LIN {X 0,Y 438.323,Z 588.239,A -85,B 0,C 180,E1 -9180.919,E2 -9180.919} C_VEL
LIN {X 0,Y 438.374,Z 587.567,A -85,B 0,C 180,E1 -9181.838,E2 -9181.838} C_VEL
LIN {X 0,Y 438.437,Z 586.498,A -85,B 0,C 180,E1 -9182.756,E2 -9182.756} C_VEL
LIN {X 0,Y 438.522,Z 585.021,A -85,B 0,C 180,E1 -9183.676,E2 -9183.676} C_VEL
LIN {X 0,Y 438.511,Z 581.969,A -85,B 0,C 180,E1 -9185.057,E2 -9185.057} C_VEL
LIN {X 0,Y 438.764,Z 577.857,A -85,B 0,C 180,E1 -9186.438,E2 -9186.438} C_VEL
LIN {X 0,Y 438.979,Z 571.563,A -85,B 0,C 180,E1 -9188.053,E2 -9188.053} C_VEL
LIN {X 0,Y 439.405,Z 564.723,A -85,B 0,C 180,E1 -9189.436,E2 -9189.436} C_VEL
LIN {X 0,Y 439.856,Z 556.275,A -85,B 0,C 180,E1 -9190.821,E2 -9190.821} C_VEL
LIN {X 0,Y 440.371,Z 547.631,A -85,B 0,C 180,E1 -9191.974,E2 -9191.974} C_VEL
LIN {X 0,Y 441.064,Z 537.577,A -85,B 0,C 180,E1 -9193.073,E2 -9193.073} C_VEL
LIN {X 0,Y 441.606,Z 526.721,A -85,B 0,C 180,E1 -9194.046,E2 -9194.046} C_VEL
LIN {X 0,Y 442.181,Z 515.563,A -85,B 0,C 180,E1 -9194.85,E2 -9194.85} C_VEL
LIN {X 0,Y 442.721,Z 503.226,A -85,B 0,C 180,E1 -9195.538,E2 -9195.538} C_VEL
LIN {X 0,Y 441.9,Z 496.755,A -85,B 0,C 180,E1 -9195.864,E2 -9195.864} C_VEL
LIN {X 0,Y 439.098,Z 483.193,A -85,B 0,C 180,E1 -9196.446,E2 -9196.446} C_VEL
LIN {X 0,Y 438.675,Z 481.043,A -85,B 0,C 180,E1 -9196.533,E2 -9196.533} C_VEL
LIN {X 0,Y 438.78,Z 475.256,A -85,B 0,C 180,E1 -9199.655,E2 -9199.655} C_VEL
LIN {X 0,Y 438.918,Z 469.873,A -85,B 0,C 180,E1 -9202.6,E2 -9202.6} C_VEL
LIN {X 0,Y 439.082,Z 464.477,A -85,B 0,C 180,E1 -9205.605,E2 -9205.605} C_VEL
LIN {X 0,Y 439.285,Z 459.037,A -85,B 0,C 180,E1 -9208.683,E2 -9208.683} C_VEL
LIN {X 0,Y 439.494,Z 453.542,A -85,B 0,C 180,E1 -9211.851,E2 -9211.851} C_VEL
LIN {X 0,Y 439.619,Z 449.852,A -85,B 0,C 180,E1 -9214.024,E2 -9214.024} C_VEL
LIN {X 0,Y 439.631,Z 446.118,A -85,B 0,C 180,E1 -9216.263,E2 -9216.263} C_VEL
LIN {X 0,Y 439.451,Z 444.373,A -85,B 0,C 180,E1 -9217.425,E2 -9217.425} C_VEL
LIN {X 0,Y 439.412,Z 444.375,A -85,B 0,C 180,E1 -9219.85,E2 -9219.85} C_VEL
LIN {X 0,Y 439.391,Z 444.378,A -85,B 0,C 180,E1 -9222.627,E2 -9222.627} C_VEL
LIN {X 0,Y 439.408,Z 444.38,A -85,B 0,C 180,E1 -9225.271,E2 -9225.271} C_VEL
LIN {X 0,Y 439.404,Z 444.38,A -85,B 0,C 180,E1 -9228.741,E2 -9228.741} C_VEL
LIN {X 0,Y 439.489,Z 444.514,A -85,B 0,C 180,E1 -9229.915,E2 -9229.915} C_VEL
LIN {X 0,Y 440.084,Z 449.479,A -85,B 0,C 180,E1 -9232.078,E2 -9232.078} C_VEL
LIN {X 0,Y 439.9,Z 456.078,A -85,B 0,C 180,E1 -9234.889,E2 -9234.889} C_VEL
LIN {X 0,Y 439.732,Z 463.121,A -85,B 0,C 180,E1 -9237.895,E2 -9237.895} C_VEL
LIN {X 0,Y 439.576,Z 469.949,A -85,B 0,C 180,E1 -9240.814,E2 -9240.814} C_VEL
LIN {X 0,Y 439.393,Z 476.574,A -85,B 0,C 180,E1 -9243.6,E2 -9243.6} C_VEL
LIN {X 0,Y 439.22,Z 483.432,A -85,B 0,C 180,E1 -9246.419,E2 -9246.419} C_VEL
LIN {X 0,Y 439.101,Z 490.898,A -85,B 0,C 180,E1 -9249.382,E2 -9249.382} C_VEL
LIN {X 0,Y 439.06,Z 492.954,A -85,B 0,C 180,E1 -9250.179,E2 -9250.179} C_VEL
LIN {X 0,Y 442.741,Z 508.655,A -85,B 0,C 180,E1 -9250.733,E2 -9250.733} C_VEL
LIN {X 0,Y 444.731,Z 520.009,A -85,B 0,C 180,E1 -9251.247,E2 -9251.247} C_VEL
LIN {X 0,Y 444.069,Z 533.417,A -85,B 0,C 180,E1 -9251.888,E2 -9251.888} C_VEL
LIN {X 0,Y 443.371,Z 546.477,A -85,B 0,C 180,E1 -9252.709,E2 -9252.709} C_VEL
LIN {X 0,Y 442.529,Z 558.139,A -85,B 0,C 180,E1 -9253.626,E2 -9253.626} C_VEL
LIN {X 0,Y 441.698,Z 569.986,A -85,B 0,C 180,E1 -9254.778,E2 -9254.778} C_VEL
LIN {X 0,Y 441.477,Z 572.611,A -85,B 0,C 180,E1 -9255.067,E2 -9255.067} C_VEL
LIN {X 0,Y 440.46,Z 577.049,A -85,B 0,C 180,E1 -9255.556,E2 -9255.556} C_VEL
LIN {X 0,Y 437.195,Z 584.006,A -85,B 0,C 180,E1 -9256.371,E2 -9256.371} C_VEL
LIN {X 0,Y 433.95,Z 590.468,A -85,B 0,C 180,E1 -9257.26,E2 -9257.26} C_VEL
LIN {X 0,Y 432.977,Z 594.128,A -85,B 0,C 180,E1 -9257.858,E2 -9257.858} C_VEL
LIN {X 0,Y 432.269,Z 602.417,A -85,B 0,C 180,E1 -9259.46,E2 -9259.46} C_VEL
LIN {X 0,Y 431.823,Z 609.29,A -85,B 0,C 180,E1 -9261.104,E2 -9261.104} C_VEL
LIN {X 0,Y 431.475,Z 615.452,A -85,B 0,C 180,E1 -9262.982,E2 -9262.982} C_VEL
LIN {X 0,Y 431.38,Z 618.954,A -85,B 0,C 180,E1 -9264.389,E2 -9264.389} C_VEL
LIN {X 0,Y 431.187,Z 622.376,A -85,B 0,C 180,E1 -9266.261,E2 -9266.261} C_VEL
LIN {X 0,Y 431.198,Z 624.413,A -85,B 0,C 180,E1 -9268.131,E2 -9268.131} C_VEL
LIN {X 0,Y 431.143,Z 625.119,A -85,B 0,C 180,E1 -9269.999,E2 -9269.999} C_VEL
LIN {X 0,Y 431.197,Z 624.493,A -85,B 0,C 180,E1 -9271.867,E2 -9271.867} C_VEL
LIN {X 0,Y 431.186,Z 622.523,A -85,B 0,C 180,E1 -9273.737,E2 -9273.737} C_VEL
LIN {X 0,Y 431.379,Z 619.168,A -85,B 0,C 180,E1 -9275.608,E2 -9275.608} C_VEL
LIN {X 0,Y 431.53,Z 614.329,A -85,B 0,C 180,E1 -9277.485,E2 -9277.485} C_VEL
LIN {X 0,Y 431.922,Z 607.864,A -85,B 0,C 180,E1 -9279.363,E2 -9279.363} C_VEL
LIN {X 0,Y 432.355,Z 600.66,A -85,B 0,C 180,E1 -9281.01,E2 -9281.01} C_VEL
LIN {X 0,Y 433.045,Z 593.096,A -85,B 0,C 180,E1 -9282.416,E2 -9282.416} C_VEL
LIN {X 0,Y 433.619,Z 584.184,A -85,B 0,C 180,E1 -9283.806,E2 -9283.806} C_VEL
LIN {X 0,Y 434.507,Z 573.995,A -85,B 0,C 180,E1 -9285.117,E2 -9285.117} C_VEL
LIN {X 0,Y 435.336,Z 562.966,A -85,B 0,C 180,E1 -9286.289,E2 -9286.289} C_VEL
LIN {X 0,Y 436.298,Z 550.821,A -85,B 0,C 180,E1 -9287.336,E2 -9287.336} C_VEL
LIN {X 0,Y 437.081,Z 538.305,A -85,B 0,C 180,E1 -9288.206,E2 -9288.206} C_VEL
LIN {X 0,Y 437.756,Z 524.511,A -85,B 0,C 180,E1 -9288.949,E2 -9288.949} C_VEL
LIN {X 0,Y 437.768,Z 519.177,A -85,B 0,C 180,E1 -9289.191,E2 -9289.191} C_VEL
LIN {X 0,Y 434.917,Z 504.739,A -85,B 0,C 180,E1 -9289.836,E2 -9289.836} C_VEL
LIN {X 0,Y 432.014,Z 492.976,A -85,B 0,C 180,E1 -9290.246,E2 -9290.246} C_VEL
LIN {X 0,Y 432.131,Z 486.1,A -85,B 0,C 180,E1 -9292.973,E2 -9292.973} C_VEL
LIN {X 0,Y 432.305,Z 478.646,A -85,B 0,C 180,E1 -9296.035,E2 -9296.035} C_VEL
LIN {X 0,Y 432.512,Z 472.428,A -85,B 0,C 180,E1 -9298.662,E2 -9298.662} C_VEL
LIN {X 0,Y 432.691,Z 465.079,A -85,B 0,C 180,E1 -9301.841,E2 -9301.841} C_VEL
LIN {X 0,Y 432.919,Z 457.333,A -85,B 0,C 180,E1 -9305.183,E2 -9305.183} C_VEL
LIN {X 0,Y 433.104,Z 450.634,A -85,B 0,C 180,E1 -9308.068,E2 -9308.068} C_VEL
LIN {X 0,Y 432.706,Z 446.81,A -85,B 0,C 180,E1 -9309.743,E2 -9309.743} C_VEL
LIN {X 0,Y 432.411,Z 445.251,A -85,B 0,C 180,E1 -9310.442,E2 -9310.442} C_VEL
LIN {X 0,Y 432.359,Z 445.256,A -85,B 0,C 180,E1 -9313.054,E2 -9313.054} C_VEL
LIN {X 0,Y 432.371,Z 445.254,A -85,B 0,C 180,E1 -9315.657,E2 -9315.657} C_VEL
LIN {X 0,Y 432.366,Z 445.254,A -85,B 0,C 180,E1 -9318.391,E2 -9318.391} C_VEL
LIN {X 0,Y 432.344,Z 445.254,A -85,B 0,C 180,E1 -9321.851,E2 -9321.851} C_VEL
LIN {X 0,Y 432.332,Z 445.253,A -85,B 0,C 180,E1 -9325.322,E2 -9325.322} C_VEL
LIN {X 0,Y 432.321,Z 445.253,A -85,B 0,C 180,E1 -9328.654,E2 -9328.654} C_VEL
LIN {X 0,Y 432.375,Z 445.251,A -85,B 0,C 180,E1 -9331.876,E2 -9331.876} C_VEL
LIN {X 0,Y 432.342,Z 445.256,A -85,B 0,C 180,E1 -9334.998,E2 -9334.998} C_VEL
LIN {X 0,Y 432.367,Z 445.244,A -85,B 0,C 180,E1 -9338.046,E2 -9338.046} C_VEL
LIN {X 0,Y 432.376,Z 445.25,A -85,B 0,C 180,E1 -9341.029,E2 -9341.029} C_VEL
LIN {X 0,Y 432.432,Z 445.246,A -85,B 0,C 180,E1 -9343.961,E2 -9343.961} C_VEL
LIN {X 0,Y 432.471,Z 445.236,A -85,B 0,C 180,E1 -9347.804,E2 -9347.804} C_VEL
LIN {X 0,Y 432.481,Z 445.234,A -85,B 0,C 180,E1 -9351.59,E2 -9351.59} C_VEL
LIN {X 0,Y 432.594,Z 445.223,A -85,B 0,C 180,E1 -9354.406,E2 -9354.406} C_VEL
LIN {X 0,Y 432.596,Z 445.221,A -85,B 0,C 180,E1 -9358.138,E2 -9358.138} C_VEL
LIN {X 0,Y 432.724,Z 445.207,A -85,B 0,C 180,E1 -9360,E2 -9360} C_VEL
LIN {X 0,Y 432.596,Z 445.214,A -85,B 0,C 180,E1 -9362.794,E2 -9362.794} C_VEL
LIN {X 0,Y 432.562,Z 445.231,A -85,B 0,C 180,E1 -9366.53,E2 -9366.53} C_VEL
LIN {X 0,Y 432.435,Z 445.24,A -85,B 0,C 180,E1 -9369.353,E2 -9369.353} C_VEL
LIN {X 0,Y 432.434,Z 445.24,A -85,B 0,C 180,E1 -9372.812,E2 -9372.812} C_VEL
LIN {X 0,Y 432.401,Z 445.242,A -85,B 0,C 180,E1 -9376.479,E2 -9376.479} C_VEL
LIN {X 0,Y 432.329,Z 445.256,A -85,B 0,C 180,E1 -9379.961,E2 -9379.961} C_VEL
LIN {X 0,Y 432.309,Z 445.257,A -85,B 0,C 180,E1 -9382.965,E2 -9382.965} C_VEL
LIN {X 0,Y 432.354,Z 445.253,A -85,B 0,C 180,E1 -9386.033,E2 -9386.033} C_VEL
LIN {X 0,Y 432.343,Z 445.257,A -85,B 0,C 180,E1 -9389.187,E2 -9389.187} C_VEL
LIN {X 0,Y 432.316,Z 445.262,A -85,B 0,C 180,E1 -9392.294,E2 -9392.294} C_VEL
LIN {X 0,Y 432.332,Z 445.257,A -85,B 0,C 180,E1 -9394.678,E2 -9394.678} C_VEL
LIN {X 0,Y 432.345,Z 445.254,A -85,B 0,C 180,E1 -9398.149,E2 -9398.149} C_VEL
LIN {X 0,Y 432.365,Z 445.251,A -85,B 0,C 180,E1 -9401.609,E2 -9401.609} C_VEL
LIN {X 0,Y 432.371,Z 445.255,A -85,B 0,C 180,E1 -9404.343,E2 -9404.343} C_VEL
LIN {X 0,Y 432.36,Z 445.255,A -85,B 0,C 180,E1 -9408.394,E2 -9408.394} C_VEL
LIN {X 0,Y 432.406,Z 445.352,A -85,B 0,C 180,E1 -9410.921,E2 -9410.921} C_VEL
LIN {X 0,Y 433.952,Z 453.805,A -85,B 0,C 180,E1 -9414.338,E2 -9414.338} C_VEL
LIN {X 0,Y 435.07,Z 459.857,A -85,B 0,C 180,E1 -9416.688,E2 -9416.688} C_VEL
LIN {X 0,Y 434.697,Z 466.214,A -85,B 0,C 180,E1 -9418.968,E2 -9418.968} C_VEL
LIN {X 0,Y 433.899,Z 476.402,A -85,B 0,C 180,E1 -9422.51,E2 -9422.51} C_VEL
LIN {X 0,Y 433.157,Z 486.96,A -85,B 0,C 180,E1 -9426.071,E2 -9426.071} C_VEL
LIN {X 0,Y 432.552,Z 497.544,A -85,B 0,C 180,E1 -9429.555,E2 -9429.555} C_VEL
LIN {X 0,Y 432.493,Z 499.108,A -85,B 0,C 180,E1 -9430.064,E2 -9430.064} C_VEL
LIN {X 0,Y 435.543,Z 514.142,A -85,B 0,C 180,E1 -9430.548,E2 -9430.548} C_VEL
LIN {X 0,Y 437.339,Z 527.333,A -85,B 0,C 180,E1 -9431.106,E2 -9431.106} C_VEL
LIN {X 0,Y 436.738,Z 540.749,A -85,B 0,C 180,E1 -9431.751,E2 -9431.751} C_VEL
LIN {X 0,Y 436.051,Z 553.155,A -85,B 0,C 180,E1 -9432.533,E2 -9432.533} C_VEL
LIN {X 0,Y 435.2,Z 565,A -85,B 0,C 180,E1 -9433.465,E2 -9433.465} C_VEL
LIN {X 0,Y 434.267,Z 576.984,A -85,B 0,C 180,E1 -9434.634,E2 -9434.634} C_VEL
LIN {X 0,Y 433.482,Z 587.773,A -85,B 0,C 180,E1 -9435.926,E2 -9435.926} C_VEL
LIN {X 0,Y 432.889,Z 595.988,A -85,B 0,C 180,E1 -9437.103,E2 -9437.103} C_VEL
LIN {X 0,Y 432.407,Z 604.261,A -85,B 0,C 180,E1 -9438.517,E2 -9438.517} C_VEL
LIN {X 0,Y 431.889,Z 612.153,A -85,B 0,C 180,E1 -9440.163,E2 -9440.163} C_VEL
LIN {X 0,Y 431.566,Z 617.671,A -85,B 0,C 180,E1 -9441.573,E2 -9441.573} C_VEL
LIN {X 0,Y 431.374,Z 623.442,A -85,B 0,C 180,E1 -9443.453,E2 -9443.453} C_VEL
LIN {X 0,Y 431.256,Z 627.631,A -85,B 0,C 180,E1 -9445.327,E2 -9445.327} C_VEL
LIN {X 0,Y 431.239,Z 630.364,A -85,B 0,C 180,E1 -9447.199,E2 -9447.199} C_VEL
LIN {X 0,Y 431.193,Z 631.718,A -85,B 0,C 180,E1 -9449.067,E2 -9449.067} C_VEL
LIN {X 0,Y 431.194,Z 631.716,A -85,B 0,C 180,E1 -9450.935,E2 -9450.935} C_VEL
LIN {X 0,Y 431.24,Z 630.356,A -85,B 0,C 180,E1 -9452.804,E2 -9452.804} C_VEL
LIN {X 0,Y 431.259,Z 627.62,A -85,B 0,C 180,E1 -9454.675,E2 -9454.675} C_VEL
LIN {X 0,Y 431.375,Z 623.432,A -85,B 0,C 180,E1 -9456.55,E2 -9456.55} C_VEL
LIN {X 0,Y 431.573,Z 617.658,A -85,B 0,C 180,E1 -9458.429,E2 -9458.429} C_VEL
LIN {X 0,Y 431.911,Z 611.127,A -85,B 0,C 180,E1 -9460.075,E2 -9460.075} C_VEL
LIN {X 0,Y 432.468,Z 602.992,A -85,B 0,C 180,E1 -9461.722,E2 -9461.722} C_VEL
LIN {X 0,Y 432.969,Z 594.448,A -85,B 0,C 180,E1 -9463.136,E2 -9463.136} C_VEL
LIN {X 0,Y 433.797,Z 584.064,A -85,B 0,C 180,E1 -9464.545,E2 -9464.545} C_VEL
LIN {X 0,Y 434.595,Z 573.594,A -85,B 0,C 180,E1 -9465.717,E2 -9465.717} C_VEL
LIN {X 0,Y 435.399,Z 562.163,A -85,B 0,C 180,E1 -9466.771,E2 -9466.771} C_VEL
LIN {X 0,Y 436.238,Z 549.602,A -85,B 0,C 180,E1 -9467.704,E2 -9467.704} C_VEL
LIN {X 0,Y 436.985,Z 535.644,A -85,B 0,C 180,E1 -9468.513,E2 -9468.513} C_VEL
LIN {X 0,Y 437.262,Z 525.796,A -85,B 0,C 180,E1 -9468.957,E2 -9468.957} C_VEL
LIN {X 0,Y 434.367,Z 506.853,A -85,B 0,C 180,E1 -9469.766,E2 -9469.766} C_VEL
LIN {X 0,Y 432.545,Z 498.491,A -85,B 0,C 180,E1 -9470.119,E2 -9470.119} C_VEL
LIN {X 0,Y 433.089,Z 488.854,A -85,B 0,C 180,E1 -9473.428,E2 -9473.428} C_VEL
LIN {X 0,Y 433.826,Z 480.569,A -85,B 0,C 180,E1 -9476.456,E2 -9476.456} C_VEL
LIN {X 0,Y 434.747,Z 472.778,A -85,B 0,C 180,E1 -9479.554,E2 -9479.554} C_VEL
LIN {X 0,Y 435.75,Z 466.846,A -85,B 0,C 180,E1 -9482.158,E2 -9482.158} C_VEL
LIN {X 0,Y 435.961,Z 463.596,A -85,B 0,C 180,E1 -9483.792,E2 -9483.792} C_VEL
LIN {X 0,Y 435.29,Z 459.741,A -85,B 0,C 180,E1 -9486.169,E2 -9486.169} C_VEL
LIN {X 0,Y 434.63,Z 456.055,A -85,B 0,C 180,E1 -9489.098,E2 -9489.098} C_VEL
LIN {X 0,Y 434.129,Z 453.741,A -85,B 0,C 180,E1 -9491.868,E2 -9491.868} C_VEL
LIN {X 0,Y 433.839,Z 452.608,A -85,B 0,C 180,E1 -9494.538,E2 -9494.538} C_VEL
LIN {X 0,Y 433.817,Z 452.479,A -85,B 0,C 180,E1 -9497.124,E2 -9497.124} C_VEL
LIN {X 0,Y 433.888,Z 453.237,A -85,B 0,C 180,E1 -9499.616,E2 -9499.616} C_VEL
LIN {X 0,Y 434.126,Z 454.981,A -85,B 0,C 180,E1 -9502.492,E2 -9502.492} C_VEL
LIN {X 0,Y 434.122,Z 456.599,A -85,B 0,C 180,E1 -9504.352,E2 -9504.352} C_VEL
LIN {X 0,Y 433.574,Z 460.031,A -85,B 0,C 180,E1 -9507.448,E2 -9507.448} C_VEL
LIN {X 0,Y 433.215,Z 463.025,A -85,B 0,C 180,E1 -9509.807,E2 -9509.807} C_VEL
LIN {X 0,Y 432.764,Z 467.893,A -85,B 0,C 180,E1 -9513.278,E2 -9513.278} C_VEL
LIN {X 0,Y 432.348,Z 473.626,A -85,B 0,C 180,E1 -9517.037,E2 -9517.037} C_VEL
LIN {X 0,Y 432.09,Z 478.453,A -85,B 0,C 180,E1 -9520.028,E2 -9520.028} C_VEL
LIN {X 0,Y 431.907,Z 482.91,A -85,B 0,C 180,E1 -9522.694,E2 -9522.694} C_VEL
LIN {X 0,Y 435.601,Z 496.817,A -85,B 0,C 180,E1 -9523.46,E2 -9523.46} C_VEL
LIN {X 0,Y 436.8,Z 504.591,A -85,B 0,C 180,E1 -9523.923,E2 -9523.923} C_VEL
LIN {X 0,Y 436.083,Z 517.539,A -85,B 0,C 180,E1 -9524.698,E2 -9524.698} C_VEL
LIN {X 0,Y 435.299,Z 529.583,A -85,B 0,C 180,E1 -9525.632,E2 -9525.632} C_VEL
LIN {X 0,Y 434.468,Z 541.516,A -85,B 0,C 180,E1 -9526.792,E2 -9526.792} C_VEL
LIN {X 0,Y 433.621,Z 552.042,A -85,B 0,C 180,E1 -9528.074,E2 -9528.074} C_VEL
LIN {X 0,Y 432.957,Z 561.383,A -85,B 0,C 180,E1 -9529.478,E2 -9529.478} C_VEL
LIN {X 0,Y 432.448,Z 568.909,A -85,B 0,C 180,E1 -9530.883,E2 -9530.883} C_VEL
LIN {X 0,Y 431.935,Z 575.885,A -85,B 0,C 180,E1 -9532.521,E2 -9532.521} C_VEL
LIN {X 0,Y 431.726,Z 580.518,A -85,B 0,C 180,E1 -9533.926,E2 -9533.926} C_VEL
LIN {X 0,Y 431.505,Z 584.058,A -85,B 0,C 180,E1 -9535.329,E2 -9535.329} C_VEL
LIN {X 0,Y 431.496,Z 585.867,A -85,B 0,C 180,E1 -9536.265,E2 -9536.265} C_VEL
LIN {X 0,Y 431.379,Z 587.216,A -85,B 0,C 180,E1 -9537.199,E2 -9537.199} C_VEL
LIN {X 0,Y 431.264,Z 588.713,A -85,B 0,C 180,E1 -9539.066,E2 -9539.066} C_VEL
LIN {X 0,Y 431.248,Z 588.865,A -85,B 0,C 180,E1 -9540,E2 -9540} C_VEL
LIN {X 0,Y 431.236,Z 588.576,A -85,B 0,C 180,E1 -9540.934,E2 -9540.934} C_VEL
LIN {X 0,Y 431.294,Z 587.886,A -85,B 0,C 180,E1 -9541.868,E2 -9541.868} C_VEL
LIN {X 0,Y 431.369,Z 586.801,A -85,B 0,C 180,E1 -9542.802,E2 -9542.802} C_VEL
LIN {X 0,Y 431.444,Z 585.302,A -85,B 0,C 180,E1 -9543.736,E2 -9543.736} C_VEL
LIN {X 0,Y 431.453,Z 582.218,A -85,B 0,C 180,E1 -9545.14,E2 -9545.14} C_VEL
LIN {X 0,Y 431.667,Z 577.501,A -85,B 0,C 180,E1 -9546.708,E2 -9546.708} C_VEL
LIN {X 0,Y 431.997,Z 570.685,A -85,B 0,C 180,E1 -9548.419,E2 -9548.419} C_VEL
LIN {X 0,Y 432.418,Z 563.565,A -85,B 0,C 180,E1 -9549.826,E2 -9549.826} C_VEL
LIN {X 0,Y 432.947,Z 554.694,A -85,B 0,C 180,E1 -9551.233,E2 -9551.233} C_VEL
LIN {X 0,Y 433.646,Z 544.694,A -85,B 0,C 180,E1 -9552.519,E2 -9552.519} C_VEL
LIN {X 0,Y 434.322,Z 534.739,A -85,B 0,C 180,E1 -9553.56,E2 -9553.56} C_VEL
LIN {X 0,Y 434.857,Z 523.63,A -85,B 0,C 180,E1 -9554.508,E2 -9554.508} C_VEL
LIN {X 0,Y 435.495,Z 511.594,A -85,B 0,C 180,E1 -9555.323,E2 -9555.323} C_VEL
LIN {X 0,Y 435.692,Z 501.751,A -85,B 0,C 180,E1 -9555.856,E2 -9555.856} C_VEL
LIN {X 0,Y 433.167,Z 488.577,A -85,B 0,C 180,E1 -9556.498,E2 -9556.498} C_VEL
LIN {X 0,Y 431.592,Z 481.162,A -85,B 0,C 180,E1 -9556.811,E2 -9556.811} C_VEL
LIN {X 0,Y 431.713,Z 475.33,A -85,B 0,C 180,E1 -9559.991,E2 -9559.991} C_VEL
LIN {X 0,Y 431.886,Z 469.92,A -85,B 0,C 180,E1 -9562.989,E2 -9562.989} C_VEL
LIN {X 0,Y 432.119,Z 463.61,A -85,B 0,C 180,E1 -9566.551,E2 -9566.551} C_VEL
LIN {X 0,Y 432.378,Z 457.191,A -85,B 0,C 180,E1 -9570.257,E2 -9570.257} C_VEL
LIN {X 0,Y 432.551,Z 451.642,A -85,B 0,C 180,E1 -9573.534,E2 -9573.534} C_VEL
LIN {X 0,Y 432.62,Z 447.905,A -85,B 0,C 180,E1 -9575.791,E2 -9575.791} C_VEL
LIN {X 0,Y 432.415,Z 445.248,A -85,B 0,C 180,E1 -9577.517,E2 -9577.517} C_VEL
LIN {X 0,Y 432.332,Z 445.257,A -85,B 0,C 180,E1 -9580.56,E2 -9580.56} C_VEL
LIN {X 0,Y 432.329,Z 445.259,A -85,B 0,C 180,E1 -9583.06,E2 -9583.06} C_VEL
LIN {X 0,Y 432.339,Z 445.26,A -85,B 0,C 180,E1 -9585.664,E2 -9585.664} C_VEL
LIN {X 0,Y 432.372,Z 445.257,A -85,B 0,C 180,E1 -9588.392,E2 -9588.392} C_VEL
LIN {X 0,Y 432.437,Z 445.4,A -85,B 0,C 180,E1 -9589.736,E2 -9589.736} C_VEL
LIN {X 0,Y 433.058,Z 450.329,A -85,B 0,C 180,E1 -9591.924,E2 -9591.924} C_VEL
LIN {X 0,Y 432.897,Z 457.046,A -85,B 0,C 180,E1 -9594.813,E2 -9594.813} C_VEL
LIN {X 0,Y 432.733,Z 463.568,A -85,B 0,C 180,E1 -9597.622,E2 -9597.622} C_VEL
LIN {X 0,Y 432.541,Z 470.988,A -85,B 0,C 180,E1 -9600.826,E2 -9600.826} C_VEL
LIN {X 0,Y 432.375,Z 477.007,A -85,B 0,C 180,E1 -9603.38,E2 -9603.38} C_VEL
LIN {X 0,Y 432.169,Z 484.596,A -85,B 0,C 180,E1 -9606.519,E2 -9606.519} C_VEL
LIN {X 0,Y 432.033,Z 492.151,A -85,B 0,C 180,E1 -9609.528,E2 -9609.528} C_VEL
LIN {X 0,Y 432.031,Z 492.973,A -85,B 0,C 180,E1 -9609.849,E2 -9609.849} C_VEL
LIN {X 0,Y 435.634,Z 508.113,A -85,B 0,C 180,E1 -9610.39,E2 -9610.39} C_VEL
LIN {X 0,Y 437.971,Z 520.738,A -85,B 0,C 180,E1 -9610.976,E2 -9610.976} C_VEL
LIN {X 0,Y 437.275,Z 534.382,A -85,B 0,C 180,E1 -9611.649,E2 -9611.649} C_VEL
LIN {X 0,Y 436.59,Z 546.521,A -85,B 0,C 180,E1 -9612.432,E2 -9612.432} C_VEL
LIN {X 0,Y 435.703,Z 558.186,A -85,B 0,C 180,E1 -9613.362,E2 -9613.362} C_VEL
LIN {X 0,Y 434.831,Z 570.037,A -85,B 0,C 180,E1 -9614.532,E2 -9614.532} C_VEL
LIN {X 0,Y 433.999,Z 579.862,A -85,B 0,C 180,E1 -9615.702,E2 -9615.702} C_VEL
LIN {X 0,Y 433.258,Z 589.648,A -85,B 0,C 180,E1 -9617.111,E2 -9617.111} C_VEL
LIN {X 0,Y 432.977,Z 594.128,A -85,B 0,C 180,E1 -9617.858,E2 -9617.858} C_VEL
LIN {X 0,Y 431.992,Z 597.662,A -85,B 0,C 180,E1 -9618.478,E2 -9618.478} C_VEL
LIN {X 0,Y 428.725,Z 603.037,A -85,B 0,C 180,E1 -9619.5,E2 -9619.5} C_VEL
LIN {X 0,Y 425.547,Z 607.883,A -85,B 0,C 180,E1 -9620.58,E2 -9620.58} C_VEL
LIN {X 0,Y 424.709,Z 610.507,A -85,B 0,C 180,E1 -9621.281,E2 -9621.281} C_VEL
LIN {X 0,Y 424.413,Z 615.508,A -85,B 0,C 180,E1 -9622.865,E2 -9622.865} C_VEL
LIN {X 0,Y 424.288,Z 619.01,A -85,B 0,C 180,E1 -9624.295,E2 -9624.295} C_VEL
LIN {X 0,Y 424.098,Z 622.432,A -85,B 0,C 180,E1 -9626.198,E2 -9626.198} C_VEL
LIN {X 0,Y 424.124,Z 624.469,A -85,B 0,C 180,E1 -9628.1,E2 -9628.1} C_VEL
LIN {X 0,Y 424.061,Z 625.174,A -85,B 0,C 180,E1 -9629.999,E2 -9629.999} C_VEL
LIN {X 0,Y 424.123,Z 624.548,A -85,B 0,C 180,E1 -9631.898,E2 -9631.898} C_VEL
LIN {X 0,Y 424.097,Z 622.578,A -85,B 0,C 180,E1 -9633.799,E2 -9633.799} C_VEL
LIN {X 0,Y 424.284,Z 619.222,A -85,B 0,C 180,E1 -9635.703,E2 -9635.703} C_VEL
LIN {X 0,Y 424.466,Z 614.382,A -85,B 0,C 180,E1 -9637.61,E2 -9637.61} C_VEL
LIN {X 0,Y 424.891,Z 607.916,A -85,B 0,C 180,E1 -9639.52,E2 -9639.52} C_VEL
LIN {X 0,Y 425.361,Z 600.71,A -85,B 0,C 180,E1 -9641.193,E2 -9641.193} C_VEL
LIN {X 0,Y 426.075,Z 593.19,A -85,B 0,C 180,E1 -9642.615,E2 -9642.615} C_VEL
LIN {X 0,Y 426.689,Z 584.072,A -85,B 0,C 180,E1 -9644.059,E2 -9644.059} C_VEL
LIN {X 0,Y 427.625,Z 574.038,A -85,B 0,C 180,E1 -9645.366,E2 -9645.366} C_VEL
LIN {X 0,Y 428.527,Z 563.005,A -85,B 0,C 180,E1 -9646.555,E2 -9646.555} C_VEL
LIN {X 0,Y 429.521,Z 550.855,A -85,B 0,C 180,E1 -9647.619,E2 -9647.619} C_VEL
LIN {X 0,Y 430.299,Z 539,A -85,B 0,C 180,E1 -9648.46,E2 -9648.46} C_VEL
LIN {X 0,Y 430.933,Z 526.371,A -85,B 0,C 180,E1 -9649.169,E2 -9649.169} C_VEL
LIN {X 0,Y 431.06,Z 520.429,A -85,B 0,C 180,E1 -9649.448,E2 -9649.448} C_VEL
LIN {X 0,Y 428.263,Z 506.294,A -85,B 0,C 180,E1 -9650.11,E2 -9650.11} C_VEL
LIN {X 0,Y 424.986,Z 492.957,A -85,B 0,C 180,E1 -9650.604,E2 -9650.604} C_VEL
LIN {X 0,Y 425.145,Z 484.759,A -85,B 0,C 180,E1 -9653.89,E2 -9653.89} C_VEL
LIN {X 0,Y 425.365,Z 477.677,A -85,B 0,C 180,E1 -9656.848,E2 -9656.848} C_VEL
LIN {X 0,Y 425.607,Z 469.802,A -85,B 0,C 180,E1 -9660.24,E2 -9660.24} C_VEL
LIN {X 0,Y 425.868,Z 460.928,A -85,B 0,C 180,E1 -9664.13,E2 -9664.13} C_VEL
LIN {X 0,Y 426.114,Z 452.807,A -85,B 0,C 180,E1 -9667.657,E2 -9667.657} C_VEL
LIN {X 0,Y 425.823,Z 448.492,A -85,B 0,C 180,E1 -9669.567,E2 -9669.567} C_VEL
LIN {X 0,Y 425.336,Z 446.133,A -85,B 0,C 180,E1 -9670.682,E2 -9670.682} C_VEL
LIN {X 0,Y 425.312,Z 446.132,A -85,B 0,C 180,E1 -9673.947,E2 -9673.947} C_VEL
LIN {X 0,Y 425.325,Z 446.133,A -85,B 0,C 180,E1 -9677.353,E2 -9677.353} C_VEL
LIN {X 0,Y 425.316,Z 446.132,A -85,B 0,C 180,E1 -9681.103,E2 -9681.103} C_VEL
LIN {X 0,Y 425.292,Z 446.135,A -85,B 0,C 180,E1 -9684.663,E2 -9684.663} C_VEL
LIN {X 0,Y 425.264,Z 446.139,A -85,B 0,C 180,E1 -9688.073,E2 -9688.073} C_VEL
LIN {X 0,Y 425.328,Z 446.131,A -85,B 0,C 180,E1 -9691.368,E2 -9691.368} C_VEL
LIN {X 0,Y 425.286,Z 446.131,A -85,B 0,C 180,E1 -9694.554,E2 -9694.554} C_VEL
LIN {X 0,Y 425.31,Z 446.122,A -85,B 0,C 180,E1 -9697.719,E2 -9697.719} C_VEL
LIN {X 0,Y 425.355,Z 446.127,A -85,B 0,C 180,E1 -9700.704,E2 -9700.704} C_VEL
LIN {X 0,Y 425.388,Z 446.124,A -85,B 0,C 180,E1 -9703.688,E2 -9703.688} C_VEL
LIN {X 0,Y 425.42,Z 446.116,A -85,B 0,C 180,E1 -9707.598,E2 -9707.598} C_VEL
LIN {X 0,Y 425.432,Z 446.112,A -85,B 0,C 180,E1 -9711.45,E2 -9711.45} C_VEL
LIN {X 0,Y 425.569,Z 446.099,A -85,B 0,C 180,E1 -9714.313,E2 -9714.313} C_VEL
LIN {X 0,Y 425.565,Z 446.097,A -85,B 0,C 180,E1 -9718.107,E2 -9718.107} C_VEL
LIN {X 0,Y 425.694,Z 446.083,A -85,B 0,C 180,E1 -9720,E2 -9720} C_VEL
LIN {X 0,Y 425.548,Z 446.09,A -85,B 0,C 180,E1 -9722.84,E2 -9722.84} C_VEL
LIN {X 0,Y 425.52,Z 446.107,A -85,B 0,C 180,E1 -9726.639,E2 -9726.639} C_VEL
LIN {X 0,Y 425.394,Z 446.115,A -85,B 0,C 180,E1 -9729.509,E2 -9729.509} C_VEL
LIN {X 0,Y 425.393,Z 446.117,A -85,B 0,C 180,E1 -9732.911,E2 -9732.911} C_VEL
LIN {X 0,Y 425.35,Z 446.118,A -85,B 0,C 180,E1 -9736.605,E2 -9736.605} C_VEL
LIN {X 0,Y 425.318,Z 446.127,A -85,B 0,C 180,E1 -9739.636,E2 -9739.636} C_VEL
LIN {X 0,Y 425.297,Z 446.133,A -85,B 0,C 180,E1 -9743.366,E2 -9743.366} C_VEL
LIN {X 0,Y 425.339,Z 446.129,A -85,B 0,C 180,E1 -9746.845,E2 -9746.845} C_VEL
LIN {X 0,Y 425.309,Z 446.131,A -85,B 0,C 180,E1 -9749.718,E2 -9749.718} C_VEL
LIN {X 0,Y 425.273,Z 446.135,A -85,B 0,C 180,E1 -9753.049,E2 -9753.049} C_VEL
LIN {X 0,Y 425.276,Z 446.137,A -85,B 0,C 180,E1 -9755.93,E2 -9755.93} C_VEL
LIN {X 0,Y 425.305,Z 446.133,A -85,B 0,C 180,E1 -9759.047,E2 -9759.047} C_VEL
LIN {X 0,Y 425.324,Z 446.133,A -85,B 0,C 180,E1 -9762.647,E2 -9762.647} C_VEL
LIN {X 0,Y 425.287,Z 446.134,A -85,B 0,C 180,E1 -9765.283,E2 -9765.283} C_VEL
LIN {X 0,Y 425.298,Z 446.135,A -85,B 0,C 180,E1 -9768.626,E2 -9768.626} C_VEL
LIN {X 0,Y 425.348,Z 446.207,A -85,B 0,C 180,E1 -9770.594,E2 -9770.594} C_VEL
LIN {X 0,Y 426.783,Z 453.952,A -85,B 0,C 180,E1 -9773.794,E2 -9773.794} C_VEL
LIN {X 0,Y 428.053,Z 460.799,A -85,B 0,C 180,E1 -9776.509,E2 -9776.509} C_VEL
LIN {X 0,Y 427.859,Z 465.644,A -85,B 0,C 180,E1 -9778.291,E2 -9778.291} C_VEL
LIN {X 0,Y 427.081,Z 474.652,A -85,B 0,C 180,E1 -9781.498,E2 -9781.498} C_VEL
LIN {X 0,Y 426.379,Z 483.677,A -85,B 0,C 180,E1 -9784.626,E2 -9784.626} C_VEL
LIN {X 0,Y 425.787,Z 492.718,A -85,B 0,C 180,E1 -9787.69,E2 -9787.69} C_VEL
LIN {X 0,Y 425.469,Z 498.754,A -85,B 0,C 180,E1 -9789.705,E2 -9789.705} C_VEL
LIN {X 0,Y 428.792,Z 515.056,A -85,B 0,C 180,E1 -9790.255,E2 -9790.255} C_VEL
LIN {X 0,Y 430.607,Z 527.96,A -85,B 0,C 180,E1 -9790.826,E2 -9790.826} C_VEL
LIN {X 0,Y 429.942,Z 541.633,A -85,B 0,C 180,E1 -9791.509,E2 -9791.509} C_VEL
LIN {X 0,Y 429.157,Z 554.699,A -85,B 0,C 180,E1 -9792.366,E2 -9792.366} C_VEL
LIN {X 0,Y 428.28,Z 566.249,A -85,B 0,C 180,E1 -9793.313,E2 -9793.313} C_VEL
LIN {X 0,Y 427.299,Z 578.008,A -85,B 0,C 180,E1 -9794.499,E2 -9794.499} C_VEL
LIN {X 0,Y 426.577,Z 587.727,A -85,B 0,C 180,E1 -9795.694,E2 -9795.694} C_VEL
LIN {X 0,Y 425.875,Z 596.548,A -85,B 0,C 180,E1 -9796.986,E2 -9796.986} C_VEL
LIN {X 0,Y 425.304,Z 605.441,A -85,B 0,C 180,E1 -9798.564,E2 -9798.564} C_VEL
LIN {X 0,Y 424.85,Z 612.101,A -85,B 0,C 180,E1 -9799.999,E2 -9799.999} C_VEL
LIN {X 0,Y 424.497,Z 617.618,A -85,B 0,C 180,E1 -9801.432,E2 -9801.432} C_VEL
LIN {X 0,Y 424.296,Z 623.388,A -85,B 0,C 180,E1 -9803.343,E2 -9803.343} C_VEL
LIN {X 0,Y 424.184,Z 627.577,A -85,B 0,C 180,E1 -9805.249,E2 -9805.249} C_VEL
LIN {X 0,Y 424.135,Z 630.308,A -85,B 0,C 180,E1 -9807.152,E2 -9807.152} C_VEL
LIN {X 0,Y 424.111,Z 631.663,A -85,B 0,C 180,E1 -9809.052,E2 -9809.052} C_VEL
LIN {X 0,Y 424.112,Z 631.66,A -85,B 0,C 180,E1 -9810.951,E2 -9810.951} C_VEL
LIN {X 0,Y 424.135,Z 630.3,A -85,B 0,C 180,E1 -9812.851,E2 -9812.851} C_VEL
LIN {X 0,Y 424.186,Z 627.564,A -85,B 0,C 180,E1 -9814.753,E2 -9814.753} C_VEL
LIN {X 0,Y 424.298,Z 623.376,A -85,B 0,C 180,E1 -9816.659,E2 -9816.659} C_VEL
LIN {X 0,Y 424.504,Z 617.603,A -85,B 0,C 180,E1 -9818.57,E2 -9818.57} C_VEL
LIN {X 0,Y 424.87,Z 611.072,A -85,B 0,C 180,E1 -9820.244,E2 -9820.244} C_VEL
LIN {X 0,Y 425.482,Z 602.939,A -85,B 0,C 180,E1 -9821.917,E2 -9821.917} C_VEL
LIN {X 0,Y 426.018,Z 594.396,A -85,B 0,C 180,E1 -9823.355,E2 -9823.355} C_VEL
LIN {X 0,Y 426.907,Z 584.014,A -85,B 0,C 180,E1 -9824.785,E2 -9824.785} C_VEL
LIN {X 0,Y 427.709,Z 573.545,A -85,B 0,C 180,E1 -9825.977,E2 -9825.977} C_VEL
LIN {X 0,Y 428.59,Z 562.118,A -85,B 0,C 180,E1 -9827.046,E2 -9827.046} C_VEL
LIN {X 0,Y 429.457,Z 549.563,A -85,B 0,C 180,E1 -9827.993,E2 -9827.993} C_VEL
LIN {X 0,Y 430.243,Z 535.921,A -85,B 0,C 180,E1 -9828.797,E2 -9828.797} C_VEL
LIN {X 0,Y 430.514,Z 526.902,A -85,B 0,C 180,E1 -9829.219,E2 -9829.219} C_VEL
LIN {X 0,Y 428.003,Z 509.246,A -85,B 0,C 180,E1 -9830.032,E2 -9830.032} C_VEL
LIN {X 0,Y 425.574,Z 498.31,A -85,B 0,C 180,E1 -9830.52,E2 -9830.52} C_VEL
LIN {X 0,Y 426.169,Z 488.964,A -85,B 0,C 180,E1 -9833.832,E2 -9833.832} C_VEL
LIN {X 0,Y 427.075,Z 479.843,A -85,B 0,C 180,E1 -9837.298,E2 -9837.298} C_VEL
LIN {X 0,Y 427.968,Z 473.214,A -85,B 0,C 180,E1 -9840.058,E2 -9840.058} C_VEL
LIN {X 0,Y 428.827,Z 468.533,A -85,B 0,C 180,E1 -9842.185,E2 -9842.185} C_VEL
LIN {X 0,Y 429.09,Z 465.332,A -85,B 0,C 180,E1 -9843.841,E2 -9843.841} C_VEL
LIN {X 0,Y 428.385,Z 461.19,A -85,B 0,C 180,E1 -9846.497,E2 -9846.497} C_VEL
LIN {X 0,Y 427.736,Z 457.718,A -85,B 0,C 180,E1 -9849.444,E2 -9849.444} C_VEL
LIN {X 0,Y 427.303,Z 455.552,A -85,B 0,C 180,E1 -9852.258,E2 -9852.258} C_VEL
LIN {X 0,Y 427.01,Z 454.544,A -85,B 0,C 180,E1 -9855.051,E2 -9855.051} C_VEL
LIN {X 0,Y 426.994,Z 454.575,A -85,B 0,C 180,E1 -9857.789,E2 -9857.789} C_VEL
LIN {X 0,Y 427.108,Z 455.622,A -85,B 0,C 180,E1 -9860.659,E2 -9860.659} C_VEL
LIN {X 0,Y 427.25,Z 456.78,A -85,B 0,C 180,E1 -9862.51,E2 -9862.51} C_VEL
LIN {X 0,Y 427.109,Z 458.784,A -85,B 0,C 180,E1 -9864.836,E2 -9864.836} C_VEL
LIN {X 0,Y 426.52,Z 462.468,A -85,B 0,C 180,E1 -9868.178,E2 -9868.178} C_VEL
LIN {X 0,Y 426.033,Z 466.624,A -85,B 0,C 180,E1 -9871.419,E2 -9871.419} C_VEL
LIN {X 0,Y 425.585,Z 471.101,A -85,B 0,C 180,E1 -9874.573,E2 -9874.573} C_VEL
LIN {X 0,Y 425.309,Z 475.867,A -85,B 0,C 180,E1 -9877.726,E2 -9877.726} C_VEL
LIN {X 0,Y 425.045,Z 480.591,A -85,B 0,C 180,E1 -9880.689,E2 -9880.689} C_VEL
LIN {X 0,Y 424.885,Z 483.229,A -85,B 0,C 180,E1 -9882.287,E2 -9882.287} C_VEL
LIN {X 0,Y 428.802,Z 497.367,A -85,B 0,C 180,E1 -9883.101,E2 -9883.101} C_VEL
LIN {X 0,Y 430.142,Z 505.343,A -85,B 0,C 180,E1 -9883.6,E2 -9883.6} C_VEL
LIN {X 0,Y 429.34,Z 518.881,A -85,B 0,C 180,E1 -9884.452,E2 -9884.452} C_VEL
LIN {X 0,Y 428.511,Z 530.521,A -85,B 0,C 180,E1 -9885.391,E2 -9885.391} C_VEL
LIN {X 0,Y 427.719,Z 541.319,A -85,B 0,C 180,E1 -9886.459,E2 -9886.459} C_VEL
LIN {X 0,Y 426.797,Z 551.102,A -85,B 0,C 180,E1 -9887.639,E2 -9887.639} C_VEL
LIN {X 0,Y 426.171,Z 560.63,A -85,B 0,C 180,E1 -9889.068,E2 -9889.068} C_VEL
LIN {X 0,Y 425.566,Z 568.379,A -85,B 0,C 180,E1 -9890.494,E2 -9890.494} C_VEL
LIN {X 0,Y 425.059,Z 574.612,A -85,B 0,C 180,E1 -9891.921,E2 -9891.921} C_VEL
LIN {X 0,Y 424.755,Z 579.598,A -85,B 0,C 180,E1 -9893.349,E2 -9893.349} C_VEL
LIN {X 0,Y 424.42,Z 583.475,A -85,B 0,C 180,E1 -9894.775,E2 -9894.775} C_VEL
LIN {X 0,Y 424.44,Z 586.304,A -85,B 0,C 180,E1 -9896.202,E2 -9896.202} C_VEL
LIN {X 0,Y 424.314,Z 587.634,A -85,B 0,C 180,E1 -9897.152,E2 -9897.152} C_VEL
LIN {X 0,Y 424.229,Z 588.564,A -85,B 0,C 180,E1 -9898.101,E2 -9898.101} C_VEL
LIN {X 0,Y 424.179,Z 589.099,A -85,B 0,C 180,E1 -9899.051,E2 -9899.051} C_VEL
LIN {X 0,Y 424.161,Z 589.222,A -85,B 0,C 180,E1 -9900,E2 -9900} C_VEL
LIN {X 0,Y 424.217,Z 588.201,A -85,B 0,C 180,E1 -9901.899,E2 -9901.899} C_VEL
LIN {X 0,Y 424.303,Z 587.096,A -85,B 0,C 180,E1 -9902.848,E2 -9902.848} C_VEL
LIN {X 0,Y 424.351,Z 585.567,A -85,B 0,C 180,E1 -9903.799,E2 -9903.799} C_VEL
LIN {X 0,Y 424.399,Z 582.449,A -85,B 0,C 180,E1 -9905.226,E2 -9905.226} C_VEL
LIN {X 0,Y 424.59,Z 578.084,A -85,B 0,C 180,E1 -9906.706,E2 -9906.706} C_VEL
LIN {X 0,Y 424.909,Z 571.867,A -85,B 0,C 180,E1 -9908.321,E2 -9908.321} C_VEL
LIN {X 0,Y 425.333,Z 564.941,A -85,B 0,C 180,E1 -9909.751,E2 -9909.751} C_VEL
LIN {X 0,Y 425.878,Z 556.381,A -85,B 0,C 180,E1 -9911.181,E2 -9911.181} C_VEL
LIN {X 0,Y 426.457,Z 547.629,A -85,B 0,C 180,E1 -9912.371,E2 -9912.371} C_VEL
LIN {X 0,Y 427.261,Z 536.383,A -85,B 0,C 180,E1 -9913.617,E2 -9913.617} C_VEL
LIN {X 0,Y 427.9,Z 525.046,A -85,B 0,C 180,E1 -9914.627,E2 -9914.627} C_VEL
LIN {X 0,Y 428.561,Z 513.31,A -85,B 0,C 180,E1 -9915.455,E2 -9915.455} C_VEL
LIN {X 0,Y 428.811,Z 502.711,A -85,B 0,C 180,E1 -9916.056,E2 -9916.056} C_VEL
LIN {X 0,Y 426.176,Z 489.166,A -85,B 0,C 180,E1 -9916.737,E2 -9916.737} C_VEL
LIN {X 0,Y 424.539,Z 481.297,A -85,B 0,C 180,E1 -9917.067,E2 -9917.067} C_VEL
LIN {X 0,Y 424.669,Z 475.4,A -85,B 0,C 180,E1 -9920.337,E2 -9920.337} C_VEL
LIN {X 0,Y 424.853,Z 469.958,A -85,B 0,C 180,E1 -9923.392,E2 -9923.392} C_VEL
LIN {X 0,Y 425.095,Z 464.047,A -85,B 0,C 180,E1 -9926.775,E2 -9926.775} C_VEL
LIN {X 0,Y 425.276,Z 458.994,A -85,B 0,C 180,E1 -9929.721,E2 -9929.721} C_VEL
LIN {X 0,Y 425.463,Z 453.434,A -85,B 0,C 180,E1 -9933.032,E2 -9933.032} C_VEL
LIN {X 0,Y 425.582,Z 448.601,A -85,B 0,C 180,E1 -9935.983,E2 -9935.983} C_VEL
LIN {X 0,Y 425.374,Z 446.125,A -85,B 0,C 180,E1 -9937.566,E2 -9937.566} C_VEL
LIN {X 0,Y 425.282,Z 446.137,A -85,B 0,C 180,E1 -9941.378,E2 -9941.378} C_VEL
LIN {X 0,Y 425.295,Z 446.135,A -85,B 0,C 180,E1 -9944.717,E2 -9944.717} C_VEL
LIN {X 0,Y 425.321,Z 446.136,A -85,B 0,C 180,E1 -9948.038,E2 -9948.038} C_VEL
LIN {X 0,Y 425.331,Z 446.16,A -85,B 0,C 180,E1 -9949.472,E2 -9949.472} C_VEL
LIN {X 0,Y 426.058,Z 451.333,A -85,B 0,C 180,E1 -9951.787,E2 -9951.787} C_VEL
LIN {X 0,Y 425.976,Z 456.209,A -85,B 0,C 180,E1 -9953.943,E2 -9953.943} C_VEL
LIN {X 0,Y 425.775,Z 463.226,A -85,B 0,C 180,E1 -9956.994,E2 -9956.994} C_VEL
LIN {X 0,Y 425.558,Z 470.796,A -85,B 0,C 180,E1 -9960.3,E2 -9960.3} C_VEL
LIN {X 0,Y 425.327,Z 478.276,A -85,B 0,C 180,E1 -9963.503,E2 -9963.503} C_VEL
LIN {X 0,Y 425.113,Z 485.789,A -85,B 0,C 180,E1 -9966.623,E2 -9966.623} C_VEL
LIN {X 0,Y 424.99,Z 492.956,A -85,B 0,C 180,E1 -9969.493,E2 -9969.493} C_VEL
LIN {X 0,Y 428.856,Z 508.956,A -85,B 0,C 180,E1 -9970.092,E2 -9970.092} C_VEL
LIN {X 0,Y 431.123,Z 521.014,A -85,B 0,C 180,E1 -9970.673,E2 -9970.673} C_VEL
LIN {X 0,Y 430.534,Z 534.176,A -85,B 0,C 180,E1 -9971.336,E2 -9971.336} C_VEL
LIN {X 0,Y 429.82,Z 546.565,A -85,B 0,C 180,E1 -9972.146,E2 -9972.146} C_VEL
LIN {X 0,Y 428.896,Z 558.234,A -85,B 0,C 180,E1 -9973.09,E2 -9973.09} C_VEL
LIN {X 0,Y 428.041,Z 569.034,A -85,B 0,C 180,E1 -9974.158,E2 -9974.158} C_VEL
LIN {X 0,Y 427.08,Z 579.914,A -85,B 0,C 180,E1 -9975.465,E2 -9975.465} C_VEL
LIN {X 0,Y 426.276,Z 589.702,A -85,B 0,C 180,E1 -9976.896,E2 -9976.896} C_VEL
LIN {X 0,Y 425.681,Z 597.831,A -85,B 0,C 180,E1 -9978.33,E2 -9978.33} C_VEL
LIN {X 0,Y 425.039,Z 605.602,A -85,B 0,C 180,E1 -9980.001,E2 -9980.001} C_VEL
LIN {X 0,Y 424.709,Z 610.507,A -85,B 0,C 180,E1 -9981.281,E2 -9981.281} C_VEL
LIN {X 0,Y 423.907,Z 612.99,A -85,B 0,C 180,E1 -9981.997,E2 -9981.997} C_VEL
LIN {X 0,Y 419.574,Z 617.891,A -85,B 0,C 180,E1 -9983.664,E2 -9983.664} C_VEL
LIN {X 0,Y 417.522,Z 620.088,A -85,B 0,C 180,E1 -9984.67,E2 -9984.67} C_VEL
LIN {X 0,Y 417.128,Z 621.002,A -85,B 0,C 180,E1 -9985.196,E2 -9985.196} C_VEL
LIN {X 0,Y 417.019,Z 623.675,A -85,B 0,C 180,E1 -9987.101,E2 -9987.101} C_VEL
LIN {X 0,Y 416.991,Z 625.043,A -85,B 0,C 180,E1 -9989.033,E2 -9989.033} C_VEL
LIN {X 0,Y 416.991,Z 625.083,A -85,B 0,C 180,E1 -9990.964,E2 -9990.964} C_VEL
LIN {X 0,Y 417.018,Z 623.787,A -85,B 0,C 180,E1 -9992.897,E2 -9992.897} C_VEL
LIN {X 0,Y 417.132,Z 621.132,A -85,B 0,C 180,E1 -9994.831,E2 -9994.831} C_VEL
LIN {X 0,Y 417.27,Z 617.049,A -85,B 0,C 180,E1 -9996.77,E2 -9996.77} C_VEL
LIN {X 0,Y 417.599,Z 611.416,A -85,B 0,C 180,E1 -9998.711,E2 -9998.711} C_VEL
LIN {X 0,Y 418.003,Z 606.046,A -85,B 0,C 180,E1 -10000.167,E2 -10000.167} C_VEL
LIN {X 0,Y 418.679,Z 598.359,A -85,B 0,C 180,E1 -10001.865,E2 -10001.865} C_VEL
LIN {X 0,Y 419.243,Z 590.163,A -85,B 0,C 180,E1 -10003.352,E2 -10003.352} C_VEL
LIN {X 0,Y 420.145,Z 580.646,A -85,B 0,C 180,E1 -10004.778,E2 -10004.778} C_VEL
LIN {X 0,Y 421.082,Z 569.902,A -85,B 0,C 180,E1 -10006.108,E2 -10006.108} C_VEL
LIN {X 0,Y 422.131,Z 557.983,A -85,B 0,C 180,E1 -10007.312,E2 -10007.312} C_VEL
LIN {X 0,Y 423.058,Z 546.232,A -85,B 0,C 180,E1 -10008.272,E2 -10008.272} C_VEL
LIN {X 0,Y 423.908,Z 533.119,A -85,B 0,C 180,E1 -10009.124,E2 -10009.124} C_VEL
LIN {X 0,Y 424.366,Z 521.933,A -85,B 0,C 180,E1 -10009.702,E2 -10009.702} C_VEL
LIN {X 0,Y 421.713,Z 508.225,A -85,B 0,C 180,E1 -10010.377,E2 -10010.377} C_VEL
LIN {X 0,Y 417.986,Z 492.957,A -85,B 0,C 180,E1 -10010.965,E2 -10010.965} C_VEL
LIN {X 0,Y 418.146,Z 484.695,A -85,B 0,C 180,E1 -10014.312,E2 -10014.312} C_VEL
LIN {X 0,Y 418.389,Z 477.133,A -85,B 0,C 180,E1 -10017.513,E2 -10017.513} C_VEL
LIN {X 0,Y 418.576,Z 470.839,A -85,B 0,C 180,E1 -10020.244,E2 -10020.244} C_VEL
LIN {X 0,Y 418.797,Z 463.206,A -85,B 0,C 180,E1 -10023.625,E2 -10023.625} C_VEL
LIN {X 0,Y 419.02,Z 456.966,A -85,B 0,C 180,E1 -10026.382,E2 -10026.382} C_VEL
LIN {X 0,Y 419.059,Z 451.257,A -85,B 0,C 180,E1 -10028.907,E2 -10028.907} C_VEL
LIN {X 0,Y 418.304,Z 447.009,A -85,B 0,C 180,E1 -10030.936,E2 -10030.936} C_VEL
LIN {X 0,Y 418.262,Z 447.01,A -85,B 0,C 180,E1 -10033.737,E2 -10033.737} C_VEL
LIN {X 0,Y 418.276,Z 447.011,A -85,B 0,C 180,E1 -10036.457,E2 -10036.457} C_VEL
LIN {X 0,Y 418.26,Z 447.012,A -85,B 0,C 180,E1 -10039.122,E2 -10039.122} C_VEL
LIN {X 0,Y 418.23,Z 447.011,A -85,B 0,C 180,E1 -10042.164,E2 -10042.164} C_VEL
LIN {X 0,Y 418.257,Z 447.006,A -85,B 0,C 180,E1 -10045.419,E2 -10045.419} C_VEL
LIN {X 0,Y 418.212,Z 447.011,A -85,B 0,C 180,E1 -10048.604,E2 -10048.604} C_VEL
LIN {X 0,Y 418.286,Z 447.006,A -85,B 0,C 180,E1 -10051.936,E2 -10051.936} C_VEL
LIN {X 0,Y 418.28,Z 447.009,A -85,B 0,C 180,E1 -10055.162,E2 -10055.162} C_VEL
LIN {X 0,Y 418.246,Z 447.002,A -85,B 0,C 180,E1 -10058.304,E2 -10058.304} C_VEL
LIN {X 0,Y 418.275,Z 447.006,A -85,B 0,C 180,E1 -10061.383,E2 -10061.383} C_VEL
LIN {X 0,Y 418.3,Z 447.002,A -85,B 0,C 180,E1 -10064.406,E2 -10064.406} C_VEL
LIN {X 0,Y 418.36,Z 446.997,A -85,B 0,C 180,E1 -10067.386,E2 -10067.386} C_VEL
LIN {X 0,Y 418.351,Z 446.998,A -85,B 0,C 180,E1 -10070.329,E2 -10070.329} C_VEL
LIN {X 0,Y 418.485,Z 446.98,A -85,B 0,C 180,E1 -10073.249,E2 -10073.249} C_VEL
LIN {X 0,Y 418.339,Z 446.995,A -85,B 0,C 180,E1 -10075.181,E2 -10075.181} C_VEL
LIN {X 0,Y 418.535,Z 446.973,A -85,B 0,C 180,E1 -10078.075,E2 -10078.075} C_VEL
LIN {X 0,Y 418.663,Z 446.959,A -85,B 0,C 180,E1 -10080,E2 -10080} C_VEL
LIN {X 0,Y 418.502,Z 446.967,A -85,B 0,C 180,E1 -10082.888,E2 -10082.888} C_VEL
LIN {X 0,Y 418.483,Z 446.982,A -85,B 0,C 180,E1 -10086.751,E2 -10086.751} C_VEL
LIN {X 0,Y 418.35,Z 446.989,A -85,B 0,C 180,E1 -10089.671,E2 -10089.671} C_VEL
LIN {X 0,Y 418.345,Z 446.996,A -85,B 0,C 180,E1 -10093.007,E2 -10093.007} C_VEL
LIN {X 0,Y 418.302,Z 446.993,A -85,B 0,C 180,E1 -10096.736,E2 -10096.736} C_VEL
LIN {X 0,Y 418.26,Z 447.007,A -85,B 0,C 180,E1 -10099.791,E2 -10099.791} C_VEL
LIN {X 0,Y 418.228,Z 447.011,A -85,B 0,C 180,E1 -10102.737,E2 -10102.737} C_VEL
LIN {X 0,Y 418.261,Z 447.009,A -85,B 0,C 180,E1 -10105.905,E2 -10105.905} C_VEL
LIN {X 0,Y 418.265,Z 447.011,A -85,B 0,C 180,E1 -10109.162,E2 -10109.162} C_VEL
LIN {X 0,Y 418.248,Z 447.011,A -85,B 0,C 180,E1 -10112.845,E2 -10112.845} C_VEL
LIN {X 0,Y 418.24,Z 447.011,A -85,B 0,C 180,E1 -10116.24,E2 -10116.24} C_VEL
LIN {X 0,Y 418.258,Z 447.011,A -85,B 0,C 180,E1 -10119.681,E2 -10119.681} C_VEL
LIN {X 0,Y 418.277,Z 447.007,A -85,B 0,C 180,E1 -10122.331,E2 -10122.331} C_VEL
LIN {X 0,Y 418.244,Z 447.012,A -85,B 0,C 180,E1 -10125.112,E2 -10125.112} C_VEL
LIN {X 0,Y 418.249,Z 447.013,A -85,B 0,C 180,E1 -10127.77,E2 -10127.77} C_VEL
LIN {X 0,Y 418.293,Z 447.038,A -85,B 0,C 180,E1 -10130.247,E2 -10130.247} C_VEL
LIN {X 0,Y 419.708,Z 454.718,A -85,B 0,C 180,E1 -10133.491,E2 -10133.491} C_VEL
LIN {X 0,Y 420.919,Z 460.883,A -85,B 0,C 180,E1 -10135.992,E2 -10135.992} C_VEL
LIN {X 0,Y 421.129,Z 463.901,A -85,B 0,C 180,E1 -10137.156,E2 -10137.156} C_VEL
LIN {X 0,Y 420.33,Z 472.74,A -85,B 0,C 180,E1 -10140.395,E2 -10140.395} C_VEL
LIN {X 0,Y 419.573,Z 481.901,A -85,B 0,C 180,E1 -10143.65,E2 -10143.65} C_VEL
LIN {X 0,Y 418.899,Z 490.918,A -85,B 0,C 180,E1 -10146.781,E2 -10146.781} C_VEL
LIN {X 0,Y 418.455,Z 498.447,A -85,B 0,C 180,E1 -10149.349,E2 -10149.349} C_VEL
LIN {X 0,Y 421.632,Z 513.705,A -85,B 0,C 180,E1 -10149.865,E2 -10149.865} C_VEL
LIN {X 0,Y 423.781,Z 527.95,A -85,B 0,C 180,E1 -10150.505,E2 -10150.505} C_VEL
LIN {X 0,Y 423.209,Z 541.326,A -85,B 0,C 180,E1 -10151.186,E2 -10151.186} C_VEL
LIN {X 0,Y 422.388,Z 554.665,A -85,B 0,C 180,E1 -10152.074,E2 -10152.074} C_VEL
LIN {X 0,Y 421.475,Z 566.209,A -85,B 0,C 180,E1 -10153.035,E2 -10153.035} C_VEL
LIN {X 0,Y 420.459,Z 577.964,A -85,B 0,C 180,E1 -10154.241,E2 -10154.241} C_VEL
LIN {X 0,Y 419.649,Z 587.68,A -85,B 0,C 180,E1 -10155.452,E2 -10155.452} C_VEL
LIN {X 0,Y 418.869,Z 597.099,A -85,B 0,C 180,E1 -10156.864,E2 -10156.864} C_VEL
LIN {X 0,Y 418.296,Z 605.39,A -85,B 0,C 180,E1 -10158.37,E2 -10158.37} C_VEL
LIN {X 0,Y 417.793,Z 612.048,A -85,B 0,C 180,E1 -10159.828,E2 -10159.828} C_VEL
LIN {X 0,Y 417.441,Z 617.565,A -85,B 0,C 180,E1 -10161.286,E2 -10161.286} C_VEL
LIN {X 0,Y 417.227,Z 623.334,A -85,B 0,C 180,E1 -10163.23,E2 -10163.23} C_VEL
LIN {X 0,Y 417.091,Z 627.522,A -85,B 0,C 180,E1 -10165.168,E2 -10165.168} C_VEL
LIN {X 0,Y 417.031,Z 630.253,A -85,B 0,C 180,E1 -10167.103,E2 -10167.103} C_VEL
LIN {X 0,Y 417.082,Z 631.1,A -85,B 0,C 180,E1 -10168.07,E2 -10168.07} C_VEL
LIN {X 0,Y 417.003,Z 631.775,A -85,B 0,C 180,E1 -10170.001,E2 -10170.001} C_VEL
LIN {X 0,Y 417.089,Z 631.094,A -85,B 0,C 180,E1 -10171.932,E2 -10171.932} C_VEL
LIN {X 0,Y 417.024,Z 629.051,A -85,B 0,C 180,E1 -10173.866,E2 -10173.866} C_VEL
LIN {X 0,Y 417.138,Z 625.603,A -85,B 0,C 180,E1 -10175.803,E2 -10175.803} C_VEL
LIN {X 0,Y 417.288,Z 620.642,A -85,B 0,C 180,E1 -10177.745,E2 -10177.745} C_VEL
LIN {X 0,Y 417.687,Z 614.014,A -85,B 0,C 180,E1 -10179.688,E2 -10179.688} C_VEL
LIN {X 0,Y 418.215,Z 606.59,A -85,B 0,C 180,E1 -10181.389,E2 -10181.389} C_VEL
LIN {X 0,Y 418.751,Z 598.673,A -85,B 0,C 180,E1 -10182.874,E2 -10182.874} C_VEL
LIN {X 0,Y 419.524,Z 589.414,A -85,B 0,C 180,E1 -10184.307,E2 -10184.307} C_VEL
LIN {X 0,Y 420.366,Z 578.978,A -85,B 0,C 180,E1 -10185.641,E2 -10185.641} C_VEL
LIN {X 0,Y 421.373,Z 567.429,A -85,B 0,C 180,E1 -10186.847,E2 -10186.847} C_VEL
LIN {X 0,Y 422.345,Z 554.577,A -85,B 0,C 180,E1 -10187.931,E2 -10187.931} C_VEL
LIN {X 0,Y 423.278,Z 540.781,A -85,B 0,C 180,E1 -10188.842,E2 -10188.842} C_VEL
LIN {X 0,Y 423.783,Z 527.968,A -85,B 0,C 180,E1 -10189.491,E2 -10189.491} C_VEL
LIN {X 0,Y 421.589,Z 511.252,A -85,B 0,C 180,E1 -10190.332,E2 -10190.332} C_VEL
LIN {X 0,Y 418.61,Z 498.147,A -85,B 0,C 180,E1 -10190.95,E2 -10190.95} C_VEL
LIN {X 0,Y 419.262,Z 489.107,A -85,B 0,C 180,E1 -10194.249,E2 -10194.249} C_VEL
LIN {X 0,Y 420.209,Z 480.658,A -85,B 0,C 180,E1 -10197.572,E2 -10197.572} C_VEL
LIN {X 0,Y 421.466,Z 472.508,A -85,B 0,C 180,E1 -10201.128,E2 -10201.128} C_VEL
LIN {X 0,Y 422.066,Z 469.148,A -85,B 0,C 180,E1 -10202.765,E2 -10202.765} C_VEL
LIN {X 0,Y 422.213,Z 467.471,A -85,B 0,C 180,E1 -10203.666,E2 -10203.666} C_VEL
LIN {X 0,Y 421.753,Z 464.27,A -85,B 0,C 180,E1 -10205.679,E2 -10205.679} C_VEL
LIN {X 0,Y 421.149,Z 460.851,A -85,B 0,C 180,E1 -10208.342,E2 -10208.342} C_VEL
LIN {X 0,Y 420.63,Z 458.225,A -85,B 0,C 180,E1 -10211.247,E2 -10211.247} C_VEL
LIN {X 0,Y 420.261,Z 456.821,A -85,B 0,C 180,E1 -10214.021,E2 -10214.021} C_VEL
LIN {X 0,Y 420.151,Z 456.43,A -85,B 0,C 180,E1 -10216.7,E2 -10216.7} C_VEL
LIN {X 0,Y 420.221,Z 456.916,A -85,B 0,C 180,E1 -10219.288,E2 -10219.288} C_VEL
LIN {X 0,Y 420.324,Z 458.128,A -85,B 0,C 180,E1 -10221.802,E2 -10221.802} C_VEL
LIN {X 0,Y 420.294,Z 459.896,A -85,B 0,C 180,E1 -10224.179,E2 -10224.179} C_VEL
LIN {X 0,Y 419.824,Z 462.516,A -85,B 0,C 180,E1 -10226.828,E2 -10226.828} C_VEL
LIN {X 0,Y 419.294,Z 465.991,A -85,B 0,C 180,E1 -10229.812,E2 -10229.812} C_VEL
LIN {X 0,Y 418.826,Z 470.267,A -85,B 0,C 180,E1 -10233.059,E2 -10233.059} C_VEL
LIN {X 0,Y 418.405,Z 474.805,A -85,B 0,C 180,E1 -10236.226,E2 -10236.226} C_VEL
LIN {X 0,Y 418.111,Z 479.527,A -85,B 0,C 180,E1 -10239.33,E2 -10239.33} C_VEL
LIN {X 0,Y 417.869,Z 483.522,A -85,B 0,C 180,E1 -10241.835,E2 -10241.835} C_VEL
LIN {X 0,Y 421.777,Z 497.117,A -85,B 0,C 180,E1 -10242.666,E2 -10242.666} C_VEL
LIN {X 0,Y 423.542,Z 506.794,A -85,B 0,C 180,E1 -10243.31,E2 -10243.31} C_VEL
LIN {X 0,Y 422.742,Z 518.769,A -85,B 0,C 180,E1 -10244.079,E2 -10244.079} C_VEL
LIN {X 0,Y 421.871,Z 530.348,A -85,B 0,C 180,E1 -10245.022,E2 -10245.022} C_VEL
LIN {X 0,Y 421,Z 541.228,A -85,B 0,C 180,E1 -10246.115,E2 -10246.115} C_VEL
LIN {X 0,Y 420.176,Z 550.131,A -85,B 0,C 180,E1 -10247.196,E2 -10247.196} C_VEL
LIN {X 0,Y 419.366,Z 559.894,A -85,B 0,C 180,E1 -10248.644,E2 -10248.644} C_VEL
LIN {X 0,Y 418.712,Z 567.834,A -85,B 0,C 180,E1 -10250.093,E2 -10250.093} C_VEL
LIN {X 0,Y 418.182,Z 573.278,A -85,B 0,C 180,E1 -10251.3,E2 -10251.3} C_VEL
LIN {X 0,Y 417.732,Z 579.56,A -85,B 0,C 180,E1 -10253.043,E2 -10253.043} C_VEL
LIN {X 0,Y 417.369,Z 583.952,A -85,B 0,C 180,E1 -10254.686,E2 -10254.686} C_VEL
LIN {X 0,Y 417.384,Z 586.737,A -85,B 0,C 180,E1 -10256.138,E2 -10256.138} C_VEL
LIN {X 0,Y 417.252,Z 588.052,A -85,B 0,C 180,E1 -10257.104,E2 -10257.104} C_VEL
LIN {X 0,Y 417.154,Z 588.966,A -85,B 0,C 180,E1 -10258.069,E2 -10258.069} C_VEL
LIN {X 0,Y 417.097,Z 589.484,A -85,B 0,C 180,E1 -10259.035,E2 -10259.035} C_VEL
LIN {X 0,Y 417.077,Z 589.575,A -85,B 0,C 180,E1 -10260,E2 -10260} C_VEL
LIN {X 0,Y 417.073,Z 589.242,A -85,B 0,C 180,E1 -10260.966,E2 -10260.966} C_VEL
LIN {X 0,Y 417.143,Z 588.51,A -85,B 0,C 180,E1 -10261.931,E2 -10261.931} C_VEL
LIN {X 0,Y 417.238,Z 587.381,A -85,B 0,C 180,E1 -10262.897,E2 -10262.897} C_VEL
LIN {X 0,Y 417.247,Z 584.868,A -85,B 0,C 180,E1 -10264.347,E2 -10264.347} C_VEL
LIN {X 0,Y 417.43,Z 581.348,A -85,B 0,C 180,E1 -10265.798,E2 -10265.798} C_VEL
LIN {X 0,Y 417.586,Z 576.737,A -85,B 0,C 180,E1 -10267.252,E2 -10267.252} C_VEL
LIN {X 0,Y 418.009,Z 569.789,A -85,B 0,C 180,E1 -10268.947,E2 -10268.947} C_VEL
LIN {X 0,Y 418.479,Z 562.27,A -85,B 0,C 180,E1 -10270.401,E2 -10270.401} C_VEL
LIN {X 0,Y 419.143,Z 552.998,A -85,B 0,C 180,E1 -10271.853,E2 -10271.853} C_VEL
LIN {X 0,Y 419.943,Z 542.392,A -85,B 0,C 180,E1 -10273.181,E2 -10273.181} C_VEL
LIN {X 0,Y 420.616,Z 530.68,A -85,B 0,C 180,E1 -10274.368,E2 -10274.368} C_VEL
LIN {X 0,Y 421.371,Z 518.266,A -85,B 0,C 180,E1 -10275.354,E2 -10275.354} C_VEL
LIN {X 0,Y 422.03,Z 505.698,A -85,B 0,C 180,E1 -10276.135,E2 -10276.135} C_VEL
LIN {X 0,Y 420.635,Z 496.775,A -85,B 0,C 180,E1 -10276.626,E2 -10276.626} C_VEL
LIN {X 0,Y 417.805,Z 483.249,A -85,B 0,C 180,E1 -10277.239,E2 -10277.239} C_VEL
LIN {X 0,Y 417.5,Z 481.455,A -85,B 0,C 180,E1 -10277.325,E2 -10277.325} C_VEL
LIN {X 0,Y 417.622,Z 475.45,A -85,B 0,C 180,E1 -10280.696,E2 -10280.696} C_VEL
LIN {X 0,Y 417.761,Z 471.811,A -85,B 0,C 180,E1 -10282.764,E2 -10282.764} C_VEL
LIN {X 0,Y 417.962,Z 466.325,A -85,B 0,C 180,E1 -10285.925,E2 -10285.925} C_VEL
LIN {X 0,Y 418.178,Z 460.803,A -85,B 0,C 180,E1 -10289.169,E2 -10289.169} C_VEL
LIN {X 0,Y 418.388,Z 455.237,A -85,B 0,C 180,E1 -10292.516,E2 -10292.516} C_VEL
LIN {X 0,Y 418.533,Z 451.481,A -85,B 0,C 180,E1 -10294.815,E2 -10294.815} C_VEL
LIN {X 0,Y 418.403,Z 447.68,A -85,B 0,C 180,E1 -10297.207,E2 -10297.207} C_VEL
LIN {X 0,Y 418.308,Z 447.005,A -85,B 0,C 180,E1 -10297.685,E2 -10297.685} C_VEL
LIN {X 0,Y 418.229,Z 447.015,A -85,B 0,C 180,E1 -10300.947,E2 -10300.947} C_VEL
LIN {X 0,Y 418.222,Z 447.018,A -85,B 0,C 180,E1 -10303.73,E2 -10303.73} C_VEL
LIN {X 0,Y 418.215,Z 447.021,A -85,B 0,C 180,E1 -10306.448,E2 -10306.448} C_VEL
LIN {X 0,Y 418.306,Z 447.154,A -85,B 0,C 180,E1 -10309.314,E2 -10309.314} C_VEL
LIN {X 0,Y 419.045,Z 452.239,A -85,B 0,C 180,E1 -10311.643,E2 -10311.643} C_VEL
LIN {X 0,Y 418.981,Z 457.677,A -85,B 0,C 180,E1 -10314.048,E2 -10314.048} C_VEL
LIN {X 0,Y 418.745,Z 464.47,A -85,B 0,C 180,E1 -10317.053,E2 -10317.053} C_VEL
LIN {X 0,Y 418.529,Z 471.865,A -85,B 0,C 180,E1 -10320.305,E2 -10320.305} C_VEL
LIN {X 0,Y 418.293,Z 479.409,A -85,B 0,C 180,E1 -10323.56,E2 -10323.56} C_VEL
LIN {X 0,Y 418.064,Z 487.001,A -85,B 0,C 180,E1 -10326.73,E2 -10326.73} C_VEL
LIN {X 0,Y 417.98,Z 492.947,A -85,B 0,C 180,E1 -10329.128,E2 -10329.128} C_VEL
LIN {X 0,Y 421.958,Z 509.173,A -85,B 0,C 180,E1 -10329.76,E2 -10329.76} C_VEL
LIN {X 0,Y 424.386,Z 522.024,A -85,B 0,C 180,E1 -10330.397,E2 -10330.397} C_VEL
LIN {X 0,Y 423.732,Z 536.001,A -85,B 0,C 180,E1 -10331.14,E2 -10331.14} C_VEL
LIN {X 0,Y 422.935,Z 548.162,A -85,B 0,C 180,E1 -10331.97,E2 -10331.97} C_VEL
LIN {X 0,Y 421.845,Z 560.809,A -85,B 0,C 180,E1 -10333.048,E2 -10333.048} C_VEL
LIN {X 0,Y 420.932,Z 572.23,A -85,B 0,C 180,E1 -10334.256,E2 -10334.256} C_VEL
LIN {X 0,Y 420.019,Z 581.714,A -85,B 0,C 180,E1 -10335.463,E2 -10335.463} C_VEL
LIN {X 0,Y 419.281,Z 590.386,A -85,B 0,C 180,E1 -10336.78,E2 -10336.78} C_VEL
LIN {X 0,Y 418.582,Z 599.096,A -85,B 0,C 180,E1 -10338.375,E2 -10338.375} C_VEL
LIN {X 0,Y 418.041,Z 605.657,A -85,B 0,C 180,E1 -10339.832,E2 -10339.832} C_VEL
LIN {X 0,Y 417.638,Z 611.106,A -85,B 0,C 180,E1 -10341.288,E2 -10341.288} C_VEL
LIN {X 0,Y 417.272,Z 616.808,A -85,B 0,C 180,E1 -10343.228,E2 -10343.228} C_VEL
LIN {X 0,Y 417.128,Z 621.002,A -85,B 0,C 180,E1 -10345.196,E2 -10345.196} C_VEL
LIN {X 0,Y 416.36,Z 622.297,A -85,B 0,C 180,E1 -10345.985,E2 -10345.985} C_VEL
LIN {X 0,Y 413.437,Z 623.921,A -85,B 0,C 180,E1 -10347.276,E2 -10347.276} C_VEL
LIN {X 0,Y 411.021,Z 624.764,A -85,B 0,C 180,E1 -10348.325,E2 -10348.325} C_VEL
LIN {X 0,Y 409.984,Z 625.145,A -85,B 0,C 180,E1 -10349.139,E2 -10349.139} C_VEL
LIN {X 0,Y 409.898,Z 625.175,A -85,B 0,C 180,E1 -10349.416,E2 -10349.416} C_VEL
LIN {X 0,Y 409.917,Z 625.138,A -85,B 0,C 180,E1 -10350.981,E2 -10350.981} C_VEL
LIN {X 0,Y 409.917,Z 623.842,A -85,B 0,C 180,E1 -10352.947,E2 -10352.947} C_VEL
LIN {X 0,Y 410.043,Z 621.187,A -85,B 0,C 180,E1 -10354.915,E2 -10354.915} C_VEL
LIN {X 0,Y 410.193,Z 617.103,A -85,B 0,C 180,E1 -10356.887,E2 -10356.887} C_VEL
LIN {X 0,Y 410.541,Z 611.469,A -85,B 0,C 180,E1 -10358.862,E2 -10358.862} C_VEL
LIN {X 0,Y 410.984,Z 606.098,A -85,B 0,C 180,E1 -10360.342,E2 -10360.342} C_VEL
LIN {X 0,Y 411.699,Z 598.409,A -85,B 0,C 180,E1 -10362.069,E2 -10362.069} C_VEL
LIN {X 0,Y 412.436,Z 589.14,A -85,B 0,C 180,E1 -10363.761,E2 -10363.761} C_VEL
LIN {X 0,Y 413.243,Z 580.691,A -85,B 0,C 180,E1 -10365.03,E2 -10365.03} C_VEL
LIN {X 0,Y 414.249,Z 569.945,A -85,B 0,C 180,E1 -10366.381,E2 -10366.381} C_VEL
LIN {X 0,Y 415.351,Z 558.02,A -85,B 0,C 180,E1 -10367.604,E2 -10367.604} C_VEL
LIN {X 0,Y 416.323,Z 546.262,A -85,B 0,C 180,E1 -10368.579,E2 -10368.579} C_VEL
LIN {X 0,Y 417.185,Z 533.293,A -85,B 0,C 180,E1 -10369.435,E2 -10369.435} C_VEL
LIN {X 0,Y 417.564,Z 522.761,A -85,B 0,C 180,E1 -10369.996,E2 -10369.996} C_VEL
LIN {X 0,Y 414.953,Z 509.077,A -85,B 0,C 180,E1 -10370.696,E2 -10370.696} C_VEL
LIN {X 0,Y 411.257,Z 494.528,A -85,B 0,C 180,E1 -10371.28,E2 -10371.28} C_VEL
LIN {X 0,Y 410.972,Z 492.952,A -85,B 0,C 180,E1 -10371.343,E2 -10371.343} C_VEL
LIN {X 0,Y 411.191,Z 483.361,A -85,B 0,C 180,E1 -10375.294,E2 -10375.294} C_VEL
LIN {X 0,Y 411.457,Z 475.748,A -85,B 0,C 180,E1 -10378.57,E2 -10378.57} C_VEL
LIN {X 0,Y 411.665,Z 468.117,A -85,B 0,C 180,E1 -10381.952,E2 -10381.952} C_VEL
LIN {X 0,Y 411.923,Z 461.246,A -85,B 0,C 180,E1 -10385.02,E2 -10385.02} C_VEL
LIN {X 0,Y 412.125,Z 453.833,A -85,B 0,C 180,E1 -10388.331,E2 -10388.331} C_VEL
LIN {X 0,Y 411.769,Z 450.583,A -85,B 0,C 180,E1 -10389.82,E2 -10389.82} C_VEL
LIN {X 0,Y 411.255,Z 447.888,A -85,B 0,C 180,E1 -10391.159,E2 -10391.159} C_VEL
LIN {X 0,Y 411.226,Z 447.888,A -85,B 0,C 180,E1 -10394.481,E2 -10394.481} C_VEL
LIN {X 0,Y 411.226,Z 447.889,A -85,B 0,C 180,E1 -10397.295,E2 -10397.295} C_VEL
LIN {X 0,Y 411.223,Z 447.885,A -85,B 0,C 180,E1 -10400.776,E2 -10400.776} C_VEL
LIN {X 0,Y 411.191,Z 447.892,A -85,B 0,C 180,E1 -10404.47,E2 -10404.47} C_VEL
LIN {X 0,Y 411.163,Z 447.896,A -85,B 0,C 180,E1 -10408.002,E2 -10408.002} C_VEL
LIN {X 0,Y 411.215,Z 447.89,A -85,B 0,C 180,E1 -10411.41,E2 -10411.41} C_VEL
LIN {X 0,Y 411.227,Z 447.883,A -85,B 0,C 180,E1 -10414.706,E2 -10414.706} C_VEL
LIN {X 0,Y 411.221,Z 447.877,A -85,B 0,C 180,E1 -10417.914,E2 -10417.914} C_VEL
LIN {X 0,Y 411.226,Z 447.885,A -85,B 0,C 180,E1 -10421.051,E2 -10421.051} C_VEL
LIN {X 0,Y 411.252,Z 447.882,A -85,B 0,C 180,E1 -10424.132,E2 -10424.132} C_VEL
LIN {X 0,Y 411.304,Z 447.879,A -85,B 0,C 180,E1 -10427.166,E2 -10427.166} C_VEL
LIN {X 0,Y 411.299,Z 447.876,A -85,B 0,C 180,E1 -10430.161,E2 -10430.161} C_VEL
LIN {X 0,Y 411.452,Z 447.857,A -85,B 0,C 180,E1 -10433.133,E2 -10433.133} C_VEL
LIN {X 0,Y 411.31,Z 447.871,A -85,B 0,C 180,E1 -10435.099,E2 -10435.099} C_VEL
LIN {X 0,Y 411.504,Z 447.848,A -85,B 0,C 180,E1 -10438.042,E2 -10438.042} C_VEL
LIN {X 0,Y 411.633,Z 447.835,A -85,B 0,C 180,E1 -10440,E2 -10440} C_VEL
LIN {X 0,Y 411.457,Z 447.843,A -85,B 0,C 180,E1 -10442.937,E2 -10442.937} C_VEL
LIN {X 0,Y 411.45,Z 447.858,A -85,B 0,C 180,E1 -10446.867,E2 -10446.867} C_VEL
LIN {X 0,Y 411.299,Z 447.864,A -85,B 0,C 180,E1 -10449.839,E2 -10449.839} C_VEL
LIN {X 0,Y 411.303,Z 447.874,A -85,B 0,C 180,E1 -10453.11,E2 -10453.11} C_VEL
LIN {X 0,Y 411.246,Z 447.87,A -85,B 0,C 180,E1 -10456.889,E2 -10456.889} C_VEL
LIN {X 0,Y 411.22,Z 447.886,A -85,B 0,C 180,E1 -10459.987,E2 -10459.987} C_VEL
LIN {X 0,Y 411.193,Z 447.888,A -85,B 0,C 180,E1 -10463.148,E2 -10463.148} C_VEL
LIN {X 0,Y 411.228,Z 447.884,A -85,B 0,C 180,E1 -10466.382,E2 -10466.382} C_VEL
LIN {X 0,Y 411.201,Z 447.888,A -85,B 0,C 180,E1 -10469.713,E2 -10469.713} C_VEL
LIN {X 0,Y 411.197,Z 447.888,A -85,B 0,C 180,E1 -10473.157,E2 -10473.157} C_VEL
LIN {X 0,Y 411.187,Z 447.888,A -85,B 0,C 180,E1 -10476.554,E2 -10476.554} C_VEL
LIN {X 0,Y 411.22,Z 447.887,A -85,B 0,C 180,E1 -10479.732,E2 -10479.732} C_VEL
LIN {X 0,Y 411.214,Z 447.889,A -85,B 0,C 180,E1 -10483.128,E2 -10483.128} C_VEL
LIN {X 0,Y 411.164,Z 447.895,A -85,B 0,C 180,E1 -10485.882,E2 -10485.882} C_VEL
LIN {X 0,Y 411.223,Z 447.888,A -85,B 0,C 180,E1 -10489.503,E2 -10489.503} C_VEL
LIN {X 0,Y 411.255,Z 447.906,A -85,B 0,C 180,E1 -10489.926,E2 -10489.926} C_VEL
LIN {X 0,Y 412.648,Z 455.458,A -85,B 0,C 180,E1 -10493.176,E2 -10493.176} C_VEL
LIN {X 0,Y 414.046,Z 462.978,A -85,B 0,C 180,E1 -10496.276,E2 -10496.276} C_VEL
LIN {X 0,Y 414.042,Z 466.586,A -85,B 0,C 180,E1 -10497.664,E2 -10497.664} C_VEL
LIN {X 0,Y 413.133,Z 475.611,A -85,B 0,C 180,E1 -10501.001,E2 -10501.001} C_VEL
LIN {X 0,Y 412.398,Z 484.523,A -85,B 0,C 180,E1 -10504.217,E2 -10504.217} C_VEL
LIN {X 0,Y 411.758,Z 492.909,A -85,B 0,C 180,E1 -10507.174,E2 -10507.174} C_VEL
LIN {X 0,Y 411.443,Z 498.063,A -85,B 0,C 180,E1 -10508.964,E2 -10508.964} C_VEL
LIN {X 0,Y 414.758,Z 513.694,A -85,B 0,C 180,E1 -10509.515,E2 -10509.515} C_VEL
LIN {X 0,Y 416.84,Z 527.248,A -85,B 0,C 180,E1 -10510.136,E2 -10510.136} C_VEL
LIN {X 0,Y 416.998,Z 532.816,A -85,B 0,C 180,E1 -10510.416,E2 -10510.416} C_VEL
LIN {X 0,Y 416.233,Z 546.096,A -85,B 0,C 180,E1 -10511.168,E2 -10511.168} C_VEL
LIN {X 0,Y 415.221,Z 559.271,A -85,B 0,C 180,E1 -10512.136,E2 -10512.136} C_VEL
LIN {X 0,Y 414.179,Z 571.173,A -85,B 0,C 180,E1 -10513.235,E2 -10513.235} C_VEL
LIN {X 0,Y 413.21,Z 582.018,A -85,B 0,C 180,E1 -10514.463,E2 -10514.463} C_VEL
LIN {X 0,Y 412.29,Z 592.712,A -85,B 0,C 180,E1 -10515.943,E2 -10515.943} C_VEL
LIN {X 0,Y 411.614,Z 601.517,A -85,B 0,C 180,E1 -10517.428,E2 -10517.428} C_VEL
LIN {X 0,Y 411.01,Z 608.822,A -85,B 0,C 180,E1 -10518.91,E2 -10518.91} C_VEL
LIN {X 0,Y 410.508,Z 615.789,A -85,B 0,C 180,E1 -10520.641,E2 -10520.641} C_VEL
LIN {X 0,Y 410.162,Z 622.024,A -85,B 0,C 180,E1 -10522.618,E2 -10522.618} C_VEL
LIN {X 0,Y 410.057,Z 625.563,A -85,B 0,C 180,E1 -10524.099,E2 -10524.099} C_VEL
LIN {X 0,Y 409.94,Z 629.008,A -85,B 0,C 180,E1 -10526.069,E2 -10526.069} C_VEL
LIN {X 0,Y 409.99,Z 631.045,A -85,B 0,C 180,E1 -10528.037,E2 -10528.037} C_VEL
LIN {X 0,Y 409.926,Z 631.72,A -85,B 0,C 180,E1 -10530.001,E2 -10530.001} C_VEL
LIN {X 0,Y 409.997,Z 631.039,A -85,B 0,C 180,E1 -10531.966,E2 -10531.966} C_VEL
LIN {X 0,Y 409.94,Z 628.996,A -85,B 0,C 180,E1 -10533.933,E2 -10533.933} C_VEL
LIN {X 0,Y 410.059,Z 625.547,A -85,B 0,C 180,E1 -10535.904,E2 -10535.904} C_VEL
LIN {X 0,Y 410.165,Z 622.008,A -85,B 0,C 180,E1 -10537.385,E2 -10537.385} C_VEL
LIN {X 0,Y 410.517,Z 615.768,A -85,B 0,C 180,E1 -10539.361,E2 -10539.361} C_VEL
LIN {X 0,Y 410.979,Z 608.792,A -85,B 0,C 180,E1 -10541.093,E2 -10541.093} C_VEL
LIN {X 0,Y 411.591,Z 601.482,A -85,B 0,C 180,E1 -10542.576,E2 -10542.576} C_VEL
LIN {X 0,Y 412.302,Z 592.667,A -85,B 0,C 180,E1 -10544.059,E2 -10544.059} C_VEL
LIN {X 0,Y 413.293,Z 581.965,A -85,B 0,C 180,E1 -10545.536,E2 -10545.536} C_VEL
LIN {X 0,Y 414.235,Z 571.107,A -85,B 0,C 180,E1 -10546.765,E2 -10546.765} C_VEL
LIN {X 0,Y 415.269,Z 559.186,A -85,B 0,C 180,E1 -10547.864,E2 -10547.864} C_VEL
LIN {X 0,Y 416.182,Z 546.674,A -85,B 0,C 180,E1 -10548.791,E2 -10548.791} C_VEL
LIN {X 0,Y 416.96,Z 533.703,A -85,B 0,C 180,E1 -10549.538,E2 -10549.538} C_VEL
LIN {X 0,Y 416.977,Z 528.265,A -85,B 0,C 180,E1 -10549.815,E2 -10549.815} C_VEL
LIN {X 0,Y 415.252,Z 513.656,A -85,B 0,C 180,E1 -10550.623,E2 -10550.623} C_VEL
LIN {X 0,Y 412.446,Z 501.145,A -85,B 0,C 180,E1 -10551.252,E2 -10551.252} C_VEL
LIN {X 0,Y 411.632,Z 497.987,A -85,B 0,C 180,E1 -10551.405,E2 -10551.405} C_VEL
LIN {X 0,Y 412.36,Z 489.304,A -85,B 0,C 180,E1 -10554.682,E2 -10554.682} C_VEL
LIN {X 0,Y 413.339,Z 481.495,A -85,B 0,C 180,E1 -10557.852,E2 -10557.852} C_VEL
LIN {X 0,Y 414.533,Z 474.192,A -85,B 0,C 180,E1 -10561.139,E2 -10561.139} C_VEL
LIN {X 0,Y 415.288,Z 469.821,A -85,B 0,C 180,E1 -10563.368,E2 -10563.368} C_VEL
LIN {X 0,Y 414.948,Z 466.264,A -85,B 0,C 180,E1 -10565.612,E2 -10565.612} C_VEL
LIN {X 0,Y 414.259,Z 462.457,A -85,B 0,C 180,E1 -10568.703,E2 -10568.703} C_VEL
LIN {X 0,Y 413.788,Z 460.096,A -85,B 0,C 180,E1 -10571.484,E2 -10571.484} C_VEL
LIN {X 0,Y 413.435,Z 458.725,A -85,B 0,C 180,E1 -10574.442,E2 -10574.442} C_VEL
LIN {X 0,Y 413.343,Z 458.44,A -85,B 0,C 180,E1 -10577.148,E2 -10577.148} C_VEL
LIN {X 0,Y 413.382,Z 459.069,A -85,B 0,C 180,E1 -10579.913,E2 -10579.913} C_VEL
LIN {X 0,Y 413.467,Z 460.26,A -85,B 0,C 180,E1 -10582.272,E2 -10582.272} C_VEL
LIN {X 0,Y 413.333,Z 462.098,A -85,B 0,C 180,E1 -10584.703,E2 -10584.703} C_VEL
LIN {X 0,Y 412.86,Z 464.324,A -85,B 0,C 180,E1 -10586.994,E2 -10586.994} C_VEL
LIN {X 0,Y 412.244,Z 468.224,A -85,B 0,C 180,E1 -10590.397,E2 -10590.397} C_VEL
LIN {X 0,Y 411.757,Z 472.451,A -85,B 0,C 180,E1 -10593.655,E2 -10593.655} C_VEL
LIN {X 0,Y 411.338,Z 477.644,A -85,B 0,C 180,E1 -10597.315,E2 -10597.315} C_VEL
LIN {X 0,Y 410.918,Z 483.325,A -85,B 0,C 180,E1 -10601.037,E2 -10601.037} C_VEL
LIN {X 0,Y 410.912,Z 483.902,A -85,B 0,C 180,E1 -10601.357,E2 -10601.357} C_VEL
LIN {X 0,Y 414.97,Z 497.633,A -85,B 0,C 180,E1 -10602.251,E2 -10602.251} C_VEL
LIN {X 0,Y 416.764,Z 506.583,A -85,B 0,C 180,E1 -10602.878,E2 -10602.878} C_VEL
LIN {X 0,Y 416.728,Z 511.648,A -85,B 0,C 180,E1 -10603.207,E2 -10603.207} C_VEL
LIN {X 0,Y 415.751,Z 523.474,A -85,B 0,C 180,E1 -10604.056,E2 -10604.056} C_VEL
LIN {X 0,Y 414.808,Z 535.15,A -85,B 0,C 180,E1 -10605.116,E2 -10605.116} C_VEL
LIN {X 0,Y 413.846,Z 545.396,A -85,B 0,C 180,E1 -10606.246,E2 -10606.246} C_VEL
LIN {X 0,Y 412.962,Z 554.538,A -85,B 0,C 180,E1 -10607.468,E2 -10607.468} C_VEL
LIN {X 0,Y 412.162,Z 563.498,A -85,B 0,C 180,E1 -10608.94,E2 -10608.94} C_VEL
LIN {X 0,Y 411.54,Z 570.768,A -85,B 0,C 180,E1 -10610.415,E2 -10610.415} C_VEL
LIN {X 0,Y 410.899,Z 577.579,A -85,B 0,C 180,E1 -10612.136,E2 -10612.136} C_VEL
LIN {X 0,Y 410.654,Z 581.41,A -85,B 0,C 180,E1 -10613.377,E2 -10613.377} C_VEL
LIN {X 0,Y 410.285,Z 585.504,A -85,B 0,C 180,E1 -10615.087,E2 -10615.087} C_VEL
LIN {X 0,Y 410.329,Z 587.204,A -85,B 0,C 180,E1 -10616.072,E2 -10616.072} C_VEL
LIN {X 0,Y 410.193,Z 588.491,A -85,B 0,C 180,E1 -10617.054,E2 -10617.054} C_VEL
LIN {X 0,Y 410.082,Z 589.38,A -85,B 0,C 180,E1 -10618.036,E2 -10618.036} C_VEL
LIN {X 0,Y 410.018,Z 589.873,A -85,B 0,C 180,E1 -10619.018,E2 -10619.018} C_VEL
LIN {X 0,Y 409.996,Z 589.926,A -85,B 0,C 180,E1 -10620,E2 -10620} C_VEL
LIN {X 0,Y 410.072,Z 588.816,A -85,B 0,C 180,E1 -10621.964,E2 -10621.964} C_VEL
LIN {X 0,Y 410.174,Z 587.664,A -85,B 0,C 180,E1 -10622.947,E2 -10622.947} C_VEL
LIN {X 0,Y 410.165,Z 585.107,A -85,B 0,C 180,E1 -10624.422,E2 -10624.422} C_VEL
LIN {X 0,Y 410.364,Z 581.537,A -85,B 0,C 180,E1 -10625.898,E2 -10625.898} C_VEL
LIN {X 0,Y 410.535,Z 576.873,A -85,B 0,C 180,E1 -10627.377,E2 -10627.377} C_VEL
LIN {X 0,Y 410.991,Z 569.846,A -85,B 0,C 180,E1 -10629.101,E2 -10629.101} C_VEL
LIN {X 0,Y 411.477,Z 562.26,A -85,B 0,C 180,E1 -10630.58,E2 -10630.58} C_VEL
LIN {X 0,Y 412.146,Z 552.895,A -85,B 0,C 180,E1 -10632.057,E2 -10632.057} C_VEL
LIN {X 0,Y 413.003,Z 542.208,A -85,B 0,C 180,E1 -10633.406,E2 -10633.406} C_VEL
LIN {X 0,Y 413.674,Z 530.904,A -85,B 0,C 180,E1 -10634.566,E2 -10634.566} C_VEL
LIN {X 0,Y 414.398,Z 519.549,A -85,B 0,C 180,E1 -10635.493,E2 -10635.493} C_VEL
LIN {X 0,Y 415.119,Z 506.428,A -85,B 0,C 180,E1 -10636.336,E2 -10636.336} C_VEL
LIN {X 0,Y 412.991,Z 494.133,A -85,B 0,C 180,E1 -10637.026,E2 -10637.026} C_VEL
LIN {X 0,Y 410.445,Z 481.61,A -85,B 0,C 180,E1 -10637.597,E2 -10637.597} C_VEL
LIN {X 0,Y 410.594,Z 475.494,A -85,B 0,C 180,E1 -10641.067,E2 -10641.067} C_VEL
LIN {X 0,Y 410.765,Z 469.994,A -85,B 0,C 180,E1 -10644.244,E2 -10644.244} C_VEL
LIN {X 0,Y 411.018,Z 464.473,A -85,B 0,C 180,E1 -10647.495,E2 -10647.495} C_VEL
LIN {X 0,Y 411.247,Z 458.904,A -85,B 0,C 180,E1 -10650.843,E2 -10650.843} C_VEL
LIN {X 0,Y 411.475,Z 453.273,A -85,B 0,C 180,E1 -10654.308,E2 -10654.308} C_VEL
LIN {X 0,Y 411.45,Z 449.465,A -85,B 0,C 180,E1 -10656.715,E2 -10656.715} C_VEL
LIN {X 0,Y 411.249,Z 447.885,A -85,B 0,C 180,E1 -10657.813,E2 -10657.813} C_VEL
LIN {X 0,Y 411.17,Z 447.894,A -85,B 0,C 180,E1 -10661.228,E2 -10661.228} C_VEL
LIN {X 0,Y 411.185,Z 447.892,A -85,B 0,C 180,E1 -10664.489,E2 -10664.489} C_VEL
LIN {X 0,Y 411.206,Z 447.893,A -85,B 0,C 180,E1 -10668.197,E2 -10668.197} C_VEL
LIN {X 0,Y 411.264,Z 448.006,A -85,B 0,C 180,E1 -10669.087,E2 -10669.087} C_VEL
LIN {X 0,Y 411.928,Z 451.859,A -85,B 0,C 180,E1 -10670.855,E2 -10670.855} C_VEL
LIN {X 0,Y 412.088,Z 455.956,A -85,B 0,C 180,E1 -10672.739,E2 -10672.739} C_VEL
LIN {X 0,Y 411.789,Z 463.904,A -85,B 0,C 180,E1 -10676.293,E2 -10676.293} C_VEL
LIN {X 0,Y 411.559,Z 471.679,A -85,B 0,C 180,E1 -10679.75,E2 -10679.75} C_VEL
LIN {X 0,Y 411.297,Z 479.455,A -85,B 0,C 180,E1 -10683.146,E2 -10683.146} C_VEL
LIN {X 0,Y 411.063,Z 486.952,A -85,B 0,C 180,E1 -10686.309,E2 -10686.309} C_VEL
LIN {X 0,Y 410.985,Z 492.953,A -85,B 0,C 180,E1 -10688.756,E2 -10688.756} C_VEL
LIN {X 0,Y 415.008,Z 509.416,A -85,B 0,C 180,E1 -10689.414,E2 -10689.414} C_VEL
LIN {X 0,Y 417.478,Z 522.204,A -85,B 0,C 180,E1 -10690.067,E2 -10690.067} C_VEL
LIN {X 0,Y 417.642,Z 524.693,A -85,B 0,C 180,E1 -10690.203,E2 -10690.203} C_VEL
LIN {X 0,Y 416.858,Z 538.303,A -85,B 0,C 180,E1 -10690.967,E2 -10690.967} C_VEL
LIN {X 0,Y 415.95,Z 551.278,A -85,B 0,C 180,E1 -10691.911,E2 -10691.911} C_VEL
LIN {X 0,Y 414.776,Z 563.377,A -85,B 0,C 180,E1 -10693.004,E2 -10693.004} C_VEL
LIN {X 0,Y 413.851,Z 574.358,A -85,B 0,C 180,E1 -10694.233,E2 -10694.233} C_VEL
LIN {X 0,Y 412.819,Z 585.146,A -85,B 0,C 180,E1 -10695.707,E2 -10695.707} C_VEL
LIN {X 0,Y 412.108,Z 594.06,A -85,B 0,C 180,E1 -10697.19,E2 -10697.19} C_VEL
LIN {X 0,Y 411.239,Z 602.583,A -85,B 0,C 180,E1 -10698.914,E2 -10698.914} C_VEL
LIN {X 0,Y 410.687,Z 609.457,A -85,B 0,C 180,E1 -10700.643,E2 -10700.643} C_VEL
LIN {X 0,Y 410.286,Z 615.62,A -85,B 0,C 180,E1 -10702.618,E2 -10702.618} C_VEL
LIN {X 0,Y 410.123,Z 619.123,A -85,B 0,C 180,E1 -10704.097,E2 -10704.097} C_VEL
LIN {X 0,Y 409.934,Z 622.544,A -85,B 0,C 180,E1 -10706.067,E2 -10706.067} C_VEL
LIN {X 0,Y 409.962,Z 624.581,A -85,B 0,C 180,E1 -10708.034,E2 -10708.034} C_VEL
LIN {X 0,Y 409.898,Z 625.175,A -85,B 0,C 180,E1 -10709.416,E2 -10709.416} C_VEL
LIN {X 0,Y 409.212,Z 625.269,A -85,B 0,C 180,E1 -10710.236,E2 -10710.236} C_VEL
LIN {X 0,Y 406.321,Z 624.898,A -85,B 0,C 180,E1 -10711.568,E2 -10711.568} C_VEL
LIN {X 0,Y 403.903,Z 624.194,A -85,B 0,C 180,E1 -10712.641,E2 -10712.641} C_VEL
LIN {X 0,Y 402.898,Z 623.379,A -85,B 0,C 180,E1 -10713.466,E2 -10713.466} C_VEL
LIN {X 0,Y 402.833,Z 623.037,A -85,B 0,C 180,E1 -10713.745,E2 -10713.745} C_VEL
LIN {X 0,Y 402.959,Z 621.241,A -85,B 0,C 180,E1 -10715.002,E2 -10715.002} C_VEL
LIN {X 0,Y 403.134,Z 617.156,A -85,B 0,C 180,E1 -10717.008,E2 -10717.008} C_VEL
LIN {X 0,Y 403.499,Z 611.521,A -85,B 0,C 180,E1 -10719.017,E2 -10719.017} C_VEL
LIN {X 0,Y 403.944,Z 606.149,A -85,B 0,C 180,E1 -10720.525,E2 -10720.525} C_VEL
LIN {X 0,Y 404.714,Z 598.459,A -85,B 0,C 180,E1 -10722.281,E2 -10722.281} C_VEL
LIN {X 0,Y 405.45,Z 589.752,A -85,B 0,C 180,E1 -10723.904,E2 -10723.904} C_VEL
LIN {X 0,Y 406.362,Z 580.737,A -85,B 0,C 180,E1 -10725.291,E2 -10725.291} C_VEL
LIN {X 0,Y 407.424,Z 569.987,A -85,B 0,C 180,E1 -10726.664,E2 -10726.664} C_VEL
LIN {X 0,Y 408.579,Z 558.057,A -85,B 0,C 180,E1 -10727.905,E2 -10727.905} C_VEL
LIN {X 0,Y 409.597,Z 546.291,A -85,B 0,C 180,E1 -10728.895,E2 -10728.895} C_VEL
LIN {X 0,Y 410.439,Z 534.161,A -85,B 0,C 180,E1 -10729.717,E2 -10729.717} C_VEL
LIN {X 0,Y 410.824,Z 523.883,A -85,B 0,C 180,E1 -10730.28,E2 -10730.28} C_VEL
LIN {X 0,Y 408.262,Z 510.221,A -85,B 0,C 180,E1 -10731.009,E2 -10731.009} C_VEL
LIN {X 0,Y 404.619,Z 495.527,A -85,B 0,C 180,E1 -10731.625,E2 -10731.625} C_VEL
LIN {X 0,Y 403.97,Z 492.946,A -85,B 0,C 180,E1 -10731.734,E2 -10731.734} C_VEL
LIN {X 0,Y 404.176,Z 484.384,A -85,B 0,C 180,E1 -10735.284,E2 -10735.284} C_VEL
LIN {X 0,Y 404.418,Z 476.859,A -85,B 0,C 180,E1 -10738.546,E2 -10738.546} C_VEL
LIN {X 0,Y 404.619,Z 469.86,A -85,B 0,C 180,E1 -10741.668,E2 -10741.668} C_VEL
LIN {X 0,Y 404.91,Z 462.645,A -85,B 0,C 180,E1 -10744.942,E2 -10744.942} C_VEL
LIN {X 0,Y 405.144,Z 455.833,A -85,B 0,C 180,E1 -10748.009,E2 -10748.009} C_VEL
LIN {X 0,Y 404.749,Z 451.598,A -85,B 0,C 180,E1 -10749.974,E2 -10749.974} C_VEL
LIN {X 0,Y 404.186,Z 448.768,A -85,B 0,C 180,E1 -10751.355,E2 -10751.355} C_VEL
LIN {X 0,Y 404.191,Z 448.764,A -85,B 0,C 180,E1 -10754.528,E2 -10754.528} C_VEL
LIN {X 0,Y 404.204,Z 448.764,A -85,B 0,C 180,E1 -10757.304,E2 -10757.304} C_VEL
LIN {X 0,Y 404.161,Z 448.765,A -85,B 0,C 180,E1 -10759.954,E2 -10759.954} C_VEL
LIN {X 0,Y 404.132,Z 448.769,A -85,B 0,C 180,E1 -10763.123,E2 -10763.123} C_VEL
LIN {X 0,Y 404.136,Z 448.766,A -85,B 0,C 180,E1 -10766.187,E2 -10766.187} C_VEL
LIN {X 0,Y 404.154,Z 448.762,A -85,B 0,C 180,E1 -10769.715,E2 -10769.715} C_VEL
LIN {X 0,Y 404.186,Z 448.757,A -85,B 0,C 180,E1 -10773.122,E2 -10773.122} C_VEL
LIN {X 0,Y 404.162,Z 448.766,A -85,B 0,C 180,E1 -10776.425,E2 -10776.425} C_VEL
LIN {X 0,Y 404.216,Z 448.756,A -85,B 0,C 180,E1 -10779.86,E2 -10779.86} C_VEL
LIN {X 0,Y 404.208,Z 448.758,A -85,B 0,C 180,E1 -10782.991,E2 -10782.991} C_VEL
LIN {X 0,Y 404.255,Z 448.754,A -85,B 0,C 180,E1 -10786.788,E2 -10786.788} C_VEL
LIN {X 0,Y 404.262,Z 448.752,A -85,B 0,C 180,E1 -10789.988,E2 -10789.988} C_VEL
LIN {X 0,Y 404.403,Z 448.736,A -85,B 0,C 180,E1 -10793.013,E2 -10793.013} C_VEL
LIN {X 0,Y 404.282,Z 448.746,A -85,B 0,C 180,E1 -10795.013,E2 -10795.013} C_VEL
LIN {X 0,Y 404.473,Z 448.724,A -85,B 0,C 180,E1 -10798.008,E2 -10798.008} C_VEL
LIN {X 0,Y 404.602,Z 448.71,A -85,B 0,C 180,E1 -10800,E2 -10800} C_VEL
LIN {X 0,Y 404.414,Z 448.719,A -85,B 0,C 180,E1 -10802.988,E2 -10802.988} C_VEL
LIN {X 0,Y 404.401,Z 448.735,A -85,B 0,C 180,E1 -10806.987,E2 -10806.987} C_VEL
LIN {X 0,Y 404.261,Z 448.738,A -85,B 0,C 180,E1 -10810.012,E2 -10810.012} C_VEL
LIN {X 0,Y 404.255,Z 448.753,A -85,B 0,C 180,E1 -10813.212,E2 -10813.212} C_VEL
LIN {X 0,Y 404.205,Z 448.746,A -85,B 0,C 180,E1 -10817.007,E2 -10817.007} C_VEL
LIN {X 0,Y 404.176,Z 448.767,A -85,B 0,C 180,E1 -10820.351,E2 -10820.351} C_VEL
LIN {X 0,Y 404.159,Z 448.768,A -85,B 0,C 180,E1 -10823.575,E2 -10823.575} C_VEL
LIN {X 0,Y 404.173,Z 448.765,A -85,B 0,C 180,E1 -10825.767,E2 -10825.767} C_VEL
LIN {X 0,Y 404.188,Z 448.759,A -85,B 0,C 180,E1 -10828,E2 -10828} C_VEL
LIN {X 0,Y 404.133,Z 448.767,A -85,B 0,C 180,E1 -10831.56,E2 -10831.56} C_VEL
LIN {X 0,Y 404.177,Z 448.764,A -85,B 0,C 180,E1 -10835.017,E2 -10835.017} C_VEL
LIN {X 0,Y 404.156,Z 448.766,A -85,B 0,C 180,E1 -10838.757,E2 -10838.757} C_VEL
LIN {X 0,Y 404.184,Z 448.762,A -85,B 0,C 180,E1 -10841.612,E2 -10841.612} C_VEL
LIN {X 0,Y 404.181,Z 448.766,A -85,B 0,C 180,E1 -10844.53,E2 -10844.53} C_VEL
LIN {X 0,Y 404.164,Z 448.767,A -85,B 0,C 180,E1 -10847.301,E2 -10847.301} C_VEL
LIN {X 0,Y 404.213,Z 448.865,A -85,B 0,C 180,E1 -10849.637,E2 -10849.637} C_VEL
LIN {X 0,Y 405.563,Z 456.198,A -85,B 0,C 180,E1 -10852.857,E2 -10852.857} C_VEL
LIN {X 0,Y 406.999,Z 463.621,A -85,B 0,C 180,E1 -10855.982,E2 -10855.982} C_VEL
LIN {X 0,Y 407.042,Z 467.82,A -85,B 0,C 180,E1 -10857.641,E2 -10857.641} C_VEL
LIN {X 0,Y 406.252,Z 475.304,A -85,B 0,C 180,E1 -10860.461,E2 -10860.461} C_VEL
LIN {X 0,Y 405.463,Z 484.282,A -85,B 0,C 180,E1 -10863.77,E2 -10863.77} C_VEL
LIN {X 0,Y 404.743,Z 493.165,A -85,B 0,C 180,E1 -10866.97,E2 -10866.97} C_VEL
LIN {X 0,Y 404.457,Z 497.709,A -85,B 0,C 180,E1 -10868.583,E2 -10868.583} C_VEL
LIN {X 0,Y 407.851,Z 513.505,A -85,B 0,C 180,E1 -10869.146,E2 -10869.146} C_VEL
LIN {X 0,Y 409.897,Z 526.454,A -85,B 0,C 180,E1 -10869.751,E2 -10869.751} C_VEL
LIN {X 0,Y 410.373,Z 531.865,A -85,B 0,C 180,E1 -10870.039,E2 -10870.039} C_VEL
LIN {X 0,Y 409.583,Z 544.546,A -85,B 0,C 180,E1 -10870.75,E2 -10870.75} C_VEL
LIN {X 0,Y 408.617,Z 557.748,A -85,B 0,C 180,E1 -10871.708,E2 -10871.708} C_VEL
LIN {X 0,Y 407.496,Z 569.96,A -85,B 0,C 180,E1 -10872.823,E2 -10872.823} C_VEL
LIN {X 0,Y 406.541,Z 580.006,A -85,B 0,C 180,E1 -10873.944,E2 -10873.944} C_VEL
LIN {X 0,Y 405.515,Z 591.039,A -85,B 0,C 180,E1 -10875.447,E2 -10875.447} C_VEL
LIN {X 0,Y 404.683,Z 600.114,A -85,B 0,C 180,E1 -10876.953,E2 -10876.953} C_VEL
LIN {X 0,Y 404.126,Z 607.656,A -85,B 0,C 180,E1 -10878.465,E2 -10878.465} C_VEL
LIN {X 0,Y 403.609,Z 613.929,A -85,B 0,C 180,E1 -10879.973,E2 -10879.973} C_VEL
LIN {X 0,Y 403.149,Z 620.549,A -85,B 0,C 180,E1 -10881.985,E2 -10881.985} C_VEL
LIN {X 0,Y 402.985,Z 625.508,A -85,B 0,C 180,E1 -10883.995,E2 -10883.995} C_VEL
LIN {X 0,Y 402.858,Z 628.953,A -85,B 0,C 180,E1 -10886,E2 -10886} C_VEL
LIN {X 0,Y 402.886,Z 630.989,A -85,B 0,C 180,E1 -10888.002,E2 -10888.002} C_VEL
LIN {X 0,Y 402.85,Z 631.664,A -85,B 0,C 180,E1 -10890.001,E2 -10890.001} C_VEL
LIN {X 0,Y 402.892,Z 630.983,A -85,B 0,C 180,E1 -10892.001,E2 -10892.001} C_VEL
LIN {X 0,Y 402.859,Z 628.94,A -85,B 0,C 180,E1 -10894.003,E2 -10894.003} C_VEL
LIN {X 0,Y 402.987,Z 625.491,A -85,B 0,C 180,E1 -10896.008,E2 -10896.008} C_VEL
LIN {X 0,Y 403.153,Z 620.531,A -85,B 0,C 180,E1 -10898.018,E2 -10898.018} C_VEL
LIN {X 0,Y 403.608,Z 613.904,A -85,B 0,C 180,E1 -10900.029,E2 -10900.029} C_VEL
LIN {X 0,Y 404.228,Z 606.482,A -85,B 0,C 180,E1 -10901.789,E2 -10901.789} C_VEL
LIN {X 0,Y 404.865,Z 598.162,A -85,B 0,C 180,E1 -10903.394,E2 -10903.394} C_VEL
LIN {X 0,Y 405.713,Z 589.311,A -85,B 0,C 180,E1 -10904.805,E2 -10904.805} C_VEL
LIN {X 0,Y 406.695,Z 578.879,A -85,B 0,C 180,E1 -10906.181,E2 -10906.181} C_VEL
LIN {X 0,Y 407.775,Z 567.336,A -85,B 0,C 180,E1 -10907.426,E2 -10907.426} C_VEL
LIN {X 0,Y 408.839,Z 554.493,A -85,B 0,C 180,E1 -10908.544,E2 -10908.544} C_VEL
LIN {X 0,Y 409.806,Z 541.259,A -85,B 0,C 180,E1 -10909.45,E2 -10909.45} C_VEL
LIN {X 0,Y 410.424,Z 530.173,A -85,B 0,C 180,E1 -10910.087,E2 -10910.087} C_VEL
LIN {X 0,Y 408.837,Z 515.551,A -85,B 0,C 180,E1 -10910.952,E2 -10910.952} C_VEL
LIN {X 0,Y 406.067,Z 503.017,A -85,B 0,C 180,E1 -10911.636,E2 -10911.636} C_VEL
LIN {X 0,Y 404.731,Z 497.743,A -85,B 0,C 180,E1 -10911.922,E2 -10911.922} C_VEL
LIN {X 0,Y 405.661,Z 488.212,A -85,B 0,C 180,E1 -10915.667,E2 -10915.667} C_VEL
LIN {X 0,Y 406.732,Z 480.588,A -85,B 0,C 180,E1 -10918.936,E2 -10918.936} C_VEL
LIN {X 0,Y 408.11,Z 473.656,A -85,B 0,C 180,E1 -10922.267,E2 -10922.267} C_VEL
LIN {X 0,Y 408.421,Z 471.55,A -85,B 0,C 180,E1 -10923.413,E2 -10923.413} C_VEL
LIN {X 0,Y 408.024,Z 467.694,A -85,B 0,C 180,E1 -10925.948,E2 -10925.948} C_VEL
LIN {X 0,Y 407.513,Z 464.776,A -85,B 0,C 180,E1 -10928.38,E2 -10928.38} C_VEL
LIN {X 0,Y 407.054,Z 462.457,A -85,B 0,C 180,E1 -10931.004,E2 -10931.004} C_VEL
LIN {X 0,Y 406.69,Z 460.989,A -85,B 0,C 180,E1 -10933.73,E2 -10933.73} C_VEL
LIN {X 0,Y 406.517,Z 460.435,A -85,B 0,C 180,E1 -10936.563,E2 -10936.563} C_VEL
LIN {X 0,Y 406.533,Z 460.856,A -85,B 0,C 180,E1 -10939.523,E2 -10939.523} C_VEL
LIN {X 0,Y 406.601,Z 461.682,A -85,B 0,C 180,E1 -10941.519,E2 -10941.519} C_VEL
LIN {X 0,Y 406.525,Z 463.279,A -85,B 0,C 180,E1 -10944,E2 -10944} C_VEL
LIN {X 0,Y 406.091,Z 465.355,A -85,B 0,C 180,E1 -10946.371,E2 -10946.371} C_VEL
LIN {X 0,Y 405.39,Z 469.054,A -85,B 0,C 180,E1 -10949.818,E2 -10949.818} C_VEL
LIN {X 0,Y 404.862,Z 473.196,A -85,B 0,C 180,E1 -10953.171,E2 -10953.171} C_VEL
LIN {X 0,Y 404.386,Z 477.65,A -85,B 0,C 180,E1 -10956.439,E2 -10956.439} C_VEL
LIN {X 0,Y 404.041,Z 482.759,A -85,B 0,C 180,E1 -10959.935,E2 -10959.935} C_VEL
LIN {X 0,Y 403.923,Z 484.168,A -85,B 0,C 180,E1 -10960.841,E2 -10960.841} C_VEL
LIN {X 0,Y 408.197,Z 498.071,A -85,B 0,C 180,E1 -10961.804,E2 -10961.804} C_VEL
LIN {X 0,Y 410.354,Z 508.939,A -85,B 0,C 180,E1 -10962.613,E2 -10962.613} C_VEL
LIN {X 0,Y 409.506,Z 520.531,A -85,B 0,C 180,E1 -10963.422,E2 -10963.422} C_VEL
LIN {X 0,Y 408.513,Z 531.71,A -85,B 0,C 180,E1 -10964.386,E2 -10964.386} C_VEL
LIN {X 0,Y 407.535,Z 542.41,A -85,B 0,C 180,E1 -10965.519,E2 -10965.519} C_VEL
LIN {X 0,Y 406.482,Z 552.043,A -85,B 0,C 180,E1 -10966.757,E2 -10966.757} C_VEL
LIN {X 0,Y 405.552,Z 561.544,A -85,B 0,C 180,E1 -10968.251,E2 -10968.251} C_VEL
LIN {X 0,Y 404.823,Z 569.288,A -85,B 0,C 180,E1 -10969.75,E2 -10969.75} C_VEL
LIN {X 0,Y 404.229,Z 574.583,A -85,B 0,C 180,E1 -10970.998,E2 -10970.998} C_VEL
LIN {X 0,Y 403.756,Z 579.783,A -85,B 0,C 180,E1 -10972.499,E2 -10972.499} C_VEL
LIN {X 0,Y 403.433,Z 583.845,A -85,B 0,C 180,E1 -10974,E2 -10974} C_VEL
LIN {X 0,Y 403.219,Z 586.01,A -85,B 0,C 180,E1 -10975,E2 -10975} C_VEL
LIN {X 0,Y 403.274,Z 587.673,A -85,B 0,C 180,E1 -10976.003,E2 -10976.003} C_VEL
LIN {X 0,Y 403.135,Z 588.937,A -85,B 0,C 180,E1 -10977.002,E2 -10977.002} C_VEL
LIN {X 0,Y 403.013,Z 589.804,A -85,B 0,C 180,E1 -10978.001,E2 -10978.001} C_VEL
LIN {X 0,Y 402.942,Z 590.264,A -85,B 0,C 180,E1 -10979.001,E2 -10979.001} C_VEL
LIN {X 0,Y 402.917,Z 590.28,A -85,B 0,C 180,E1 -10980,E2 -10980} C_VEL
LIN {X 0,Y 403.003,Z 589.115,A -85,B 0,C 180,E1 -10981.999,E2 -10981.999} C_VEL
LIN {X 0,Y 403.092,Z 587.928,A -85,B 0,C 180,E1 -10982.998,E2 -10982.998} C_VEL
LIN {X 0,Y 403.089,Z 585.328,A -85,B 0,C 180,E1 -10984.5,E2 -10984.5} C_VEL
LIN {X 0,Y 403.3,Z 581.709,A -85,B 0,C 180,E1 -10986.002,E2 -10986.002} C_VEL
LIN {X 0,Y 403.489,Z 576.992,A -85,B 0,C 180,E1 -10987.506,E2 -10987.506} C_VEL
LIN {X 0,Y 403.978,Z 569.887,A -85,B 0,C 180,E1 -10989.261,E2 -10989.261} C_VEL
LIN {X 0,Y 404.483,Z 562.246,A -85,B 0,C 180,E1 -10990.765,E2 -10990.765} C_VEL
LIN {X 0,Y 405.041,Z 554.507,A -85,B 0,C 180,E1 -10992.018,E2 -10992.018} C_VEL
LIN {X 0,Y 405.834,Z 545.223,A -85,B 0,C 180,E1 -10993.265,E2 -10993.265} C_VEL
LIN {X 0,Y 406.585,Z 533.569,A -85,B 0,C 180,E1 -10994.534,E2 -10994.534} C_VEL
LIN {X 0,Y 407.302,Z 522.44,A -85,B 0,C 180,E1 -10995.513,E2 -10995.513} C_VEL
LIN {X 0,Y 408.043,Z 510.493,A -85,B 0,C 180,E1 -10996.346,E2 -10996.346} C_VEL
LIN {X 0,Y 408.094,Z 505.698,A -85,B 0,C 180,E1 -10996.635,E2 -10996.635} C_VEL
LIN {X 0,Y 405.406,Z 491.727,A -85,B 0,C 180,E1 -10997.417,E2 -10997.417} C_VEL
LIN {X 0,Y 403.368,Z 481.75,A -85,B 0,C 180,E1 -10997.862,E2 -10997.862} C_VEL
LIN {X 0,Y 403.54,Z 475.527,A -85,B 0,C 180,E1 -11001.453,E2 -11001.453} C_VEL
LIN {X 0,Y 403.747,Z 469.994,A -85,B 0,C 180,E1 -11004.694,E2 -11004.694} C_VEL
LIN {X 0,Y 403.983,Z 464.447,A -85,B 0,C 180,E1 -11008.016,E2 -11008.016} C_VEL
LIN {X 0,Y 404.243,Z 458.607,A -85,B 0,C 180,E1 -11011.58,E2 -11011.58} C_VEL
LIN {X 0,Y 404.458,Z 453.163,A -85,B 0,C 180,E1 -11014.989,E2 -11014.989} C_VEL
LIN {X 0,Y 404.228,Z 448.84,A -85,B 0,C 180,E1 -11017.797,E2 -11017.797} C_VEL
LIN {X 0,Y 404.125,Z 448.772,A -85,B 0,C 180,E1 -11021.365,E2 -11021.365} C_VEL
LIN {X 0,Y 404.154,Z 448.768,A -85,B 0,C 180,E1 -11024.522,E2 -11024.522} C_VEL
LIN {X 0,Y 404.177,Z 448.769,A -85,B 0,C 180,E1 -11027.3,E2 -11027.3} C_VEL
LIN {X 0,Y 404.171,Z 448.783,A -85,B 0,C 180,E1 -11028.799,E2 -11028.799} C_VEL
LIN {X 0,Y 405.047,Z 454.248,A -85,B 0,C 180,E1 -11031.343,E2 -11031.343} C_VEL
LIN {X 0,Y 405.013,Z 459.683,A -85,B 0,C 180,E1 -11033.843,E2 -11033.843} C_VEL
LIN {X 0,Y 404.739,Z 466.541,A -85,B 0,C 180,E1 -11036.942,E2 -11036.942} C_VEL
LIN {X 0,Y 404.511,Z 474.032,A -85,B 0,C 180,E1 -11040.309,E2 -11040.309} C_VEL
LIN {X 0,Y 404.218,Z 481.736,A -85,B 0,C 180,E1 -11043.68,E2 -11043.68} C_VEL
LIN {X 0,Y 404.018,Z 488.194,A -85,B 0,C 180,E1 -11046.415,E2 -11046.415} C_VEL
LIN {X 0,Y 403.964,Z 492.998,A -85,B 0,C 180,E1 -11048.385,E2 -11048.385} C_VEL
LIN {X 0,Y 407.783,Z 508.168,A -85,B 0,C 180,E1 -11048.991,E2 -11048.991} C_VEL
LIN {X 0,Y 410.341,Z 520.989,A -85,B 0,C 180,E1 -11049.647,E2 -11049.647} C_VEL
LIN {X 0,Y 410.925,Z 525.933,A -85,B 0,C 180,E1 -11049.929,E2 -11049.929} C_VEL
LIN {X 0,Y 410.113,Z 538.955,A -85,B 0,C 180,E1 -11050.684,E2 -11050.684} C_VEL
LIN {X 0,Y 409.204,Z 551.323,A -85,B 0,C 180,E1 -11051.603,E2 -11051.603} C_VEL
LIN {X 0,Y 407.993,Z 563.425,A -85,B 0,C 180,E1 -11052.713,E2 -11052.713} C_VEL
LIN {X 0,Y 407.022,Z 574.409,A -85,B 0,C 180,E1 -11053.961,E2 -11053.961} C_VEL
LIN {X 0,Y 405.916,Z 585.199,A -85,B 0,C 180,E1 -11055.459,E2 -11055.459} C_VEL
LIN {X 0,Y 405.276,Z 592.395,A -85,B 0,C 180,E1 -11056.648,E2 -11056.648} C_VEL
LIN {X 0,Y 404.488,Z 600.417,A -85,B 0,C 180,E1 -11058.219,E2 -11058.219} C_VEL
LIN {X 0,Y 403.823,Z 607.73,A -85,B 0,C 180,E1 -11059.976,E2 -11059.976} C_VEL
LIN {X 0,Y 403.309,Z 614.273,A -85,B 0,C 180,E1 -11061.985,E2 -11061.985} C_VEL
LIN {X 0,Y 403.067,Z 619.179,A -85,B 0,C 180,E1 -11063.994,E2 -11063.994} C_VEL
LIN {X 0,Y 402.856,Z 622.6,A -85,B 0,C 180,E1 -11065.997,E2 -11065.997} C_VEL
LIN {X 0,Y 402.859,Z 624.637,A -85,B 0,C 180,E1 -11067.999,E2 -11067.999} C_VEL
LIN {X 0,Y 402.831,Z 625.341,A -85,B 0,C 180,E1 -11069.999,E2 -11069.999} C_VEL
LIN {X 0,Y 402.858,Z 624.713,A -85,B 0,C 180,E1 -11071.998,E2 -11071.998} C_VEL
LIN {X 0,Y 402.833,Z 623.037,A -85,B 0,C 180,E1 -11073.745,E2 -11073.745} C_VEL
LIN {X 0,Y 402.226,Z 621.98,A -85,B 0,C 180,E1 -11074.567,E2 -11074.567} C_VEL
LIN {X 0,Y 399.469,Z 619.808,A -85,B 0,C 180,E1 -11075.894,E2 -11075.894} C_VEL
LIN {X 0,Y 397.164,Z 617.628,A -85,B 0,C 180,E1 -11076.948,E2 -11076.948} C_VEL
LIN {X 0,Y 396.242,Z 615.708,A -85,B 0,C 180,E1 -11077.749,E2 -11077.749} C_VEL
LIN {X 0,Y 396.204,Z 614.974,A -85,B 0,C 180,E1 -11078.017,E2 -11078.017} C_VEL
LIN {X 0,Y 396.604,Z 609.907,A -85,B 0,C 180,E1 -11079.69,E2 -11079.69} C_VEL
LIN {X 0,Y 397.193,Z 603.111,A -85,B 0,C 180,E1 -11081.481,E2 -11081.481} C_VEL
LIN {X 0,Y 398.074,Z 594.673,A -85,B 0,C 180,E1 -11083.267,E2 -11083.267} C_VEL
LIN {X 0,Y 398.903,Z 585.856,A -85,B 0,C 180,E1 -11084.8,E2 -11084.8} C_VEL
LIN {X 0,Y 400.109,Z 575.184,A -85,B 0,C 180,E1 -11086.321,E2 -11086.321} C_VEL
LIN {X 0,Y 401.217,Z 564.372,A -85,B 0,C 180,E1 -11087.586,E2 -11087.586} C_VEL
LIN {X 0,Y 402.36,Z 552.519,A -85,B 0,C 180,E1 -11088.719,E2 -11088.719} C_VEL
LIN {X 0,Y 403.355,Z 540.03,A -85,B 0,C 180,E1 -11089.678,E2 -11089.678} C_VEL
LIN {X 0,Y 404.123,Z 527.439,A -85,B 0,C 180,E1 -11090.441,E2 -11090.441} C_VEL
LIN {X 0,Y 404.013,Z 524.457,A -85,B 0,C 180,E1 -11090.607,E2 -11090.607} C_VEL
LIN {X 0,Y 401.543,Z 511.281,A -85,B 0,C 180,E1 -11091.335,E2 -11091.335} C_VEL
LIN {X 0,Y 397.972,Z 497.057,A -85,B 0,C 180,E1 -11091.969,E2 -11091.969} C_VEL
LIN {X 0,Y 396.956,Z 492.952,A -85,B 0,C 180,E1 -11092.137,E2 -11092.137} C_VEL
LIN {X 0,Y 397.146,Z 484.895,A -85,B 0,C 180,E1 -11095.51,E2 -11095.51} C_VEL
LIN {X 0,Y 397.403,Z 477.996,A -85,B 0,C 180,E1 -11098.52,E2 -11098.52} C_VEL
LIN {X 0,Y 397.591,Z 471.588,A -85,B 0,C 180,E1 -11101.396,E2 -11101.396} C_VEL
LIN {X 0,Y 397.921,Z 463.685,A -85,B 0,C 180,E1 -11105.028,E2 -11105.028} C_VEL
LIN {X 0,Y 398.157,Z 456.841,A -85,B 0,C 180,E1 -11108.153,E2 -11108.153} C_VEL
LIN {X 0,Y 397.79,Z 452.929,A -85,B 0,C 180,E1 -11109.991,E2 -11109.991} C_VEL
LIN {X 0,Y 397.161,Z 449.642,A -85,B 0,C 180,E1 -11111.572,E2 -11111.572} C_VEL
LIN {X 0,Y 397.144,Z 449.642,A -85,B 0,C 180,E1 -11115.058,E2 -11115.058} C_VEL
LIN {X 0,Y 397.149,Z 449.641,A -85,B 0,C 180,E1 -11118.005,E2 -11118.005} C_VEL
LIN {X 0,Y 397.102,Z 449.645,A -85,B 0,C 180,E1 -11121.725,E2 -11121.725} C_VEL
LIN {X 0,Y 397.117,Z 449.638,A -85,B 0,C 180,E1 -11125.506,E2 -11125.506} C_VEL
LIN {X 0,Y 397.082,Z 449.64,A -85,B 0,C 180,E1 -11129.118,E2 -11129.118} C_VEL
LIN {X 0,Y 397.185,Z 449.631,A -85,B 0,C 180,E1 -11132.609,E2 -11132.609} C_VEL
LIN {X 0,Y 397.125,Z 449.641,A -85,B 0,C 180,E1 -11135.981,E2 -11135.981} C_VEL
LIN {X 0,Y 397.157,Z 449.635,A -85,B 0,C 180,E1 -11139.693,E2 -11139.693} C_VEL
LIN {X 0,Y 397.173,Z 449.635,A -85,B 0,C 180,E1 -11142.843,E2 -11142.843} C_VEL
LIN {X 0,Y 397.172,Z 449.637,A -85,B 0,C 180,E1 -11145.657,E2 -11145.657} C_VEL
LIN {X 0,Y 397.201,Z 449.631,A -85,B 0,C 180,E1 -11148.777,E2 -11148.777} C_VEL
LIN {X 0,Y 397.384,Z 449.607,A -85,B 0,C 180,E1 -11152.04,E2 -11152.04} C_VEL
LIN {X 0,Y 397.254,Z 449.622,A -85,B 0,C 180,E1 -11154.925,E2 -11154.925} C_VEL
LIN {X 0,Y 397.442,Z 449.6,A -85,B 0,C 180,E1 -11157.973,E2 -11157.973} C_VEL
LIN {X 0,Y 397.572,Z 449.586,A -85,B 0,C 180,E1 -11160,E2 -11160} C_VEL
LIN {X 0,Y 397.373,Z 449.595,A -85,B 0,C 180,E1 -11163.041,E2 -11163.041} C_VEL
LIN {X 0,Y 397.353,Z 449.613,A -85,B 0,C 180,E1 -11167.112,E2 -11167.112} C_VEL
LIN {X 0,Y 397.219,Z 449.613,A -85,B 0,C 180,E1 -11170.191,E2 -11170.191} C_VEL
LIN {X 0,Y 397.215,Z 449.631,A -85,B 0,C 180,E1 -11173.321,E2 -11173.321} C_VEL
LIN {X 0,Y 397.171,Z 449.621,A -85,B 0,C 180,E1 -11177.156,E2 -11177.156} C_VEL
LIN {X 0,Y 397.103,Z 449.645,A -85,B 0,C 180,E1 -11180.73,E2 -11180.73} C_VEL
LIN {X 0,Y 397.122,Z 449.643,A -85,B 0,C 180,E1 -11184.019,E2 -11184.019} C_VEL
LIN {X 0,Y 397.185,Z 449.635,A -85,B 0,C 180,E1 -11187.391,E2 -11187.391} C_VEL
LIN {X 0,Y 397.075,Z 449.648,A -85,B 0,C 180,E1 -11190.883,E2 -11190.883} C_VEL
LIN {X 0,Y 397.117,Z 449.645,A -85,B 0,C 180,E1 -11194.494,E2 -11194.494} C_VEL
LIN {X 0,Y 397.102,Z 449.644,A -85,B 0,C 180,E1 -11198.275,E2 -11198.275} C_VEL
LIN {X 0,Y 397.148,Z 449.638,A -85,B 0,C 180,E1 -11201.994,E2 -11201.994} C_VEL
LIN {X 0,Y 397.103,Z 449.646,A -85,B 0,C 180,E1 -11205.067,E2 -11205.067} C_VEL
LIN {X 0,Y 397.103,Z 449.648,A -85,B 0,C 180,E1 -11208.015,E2 -11208.015} C_VEL
LIN {X 0,Y 397.169,Z 449.737,A -85,B 0,C 180,E1 -11209.302,E2 -11209.302} C_VEL
LIN {X 0,Y 398.497,Z 456.899,A -85,B 0,C 180,E1 -11212.526,E2 -11212.526} C_VEL
LIN {X 0,Y 399.962,Z 464.498,A -85,B 0,C 180,E1 -11215.787,E2 -11215.787} C_VEL
LIN {X 0,Y 400.086,Z 468.692,A -85,B 0,C 180,E1 -11217.477,E2 -11217.477} C_VEL
LIN {X 0,Y 399.235,Z 476.471,A -85,B 0,C 180,E1 -11220.47,E2 -11220.47} C_VEL
LIN {X 0,Y 398.412,Z 485.433,A -85,B 0,C 180,E1 -11223.834,E2 -11223.834} C_VEL
LIN {X 0,Y 397.649,Z 494.39,A -85,B 0,C 180,E1 -11227.12,E2 -11227.12} C_VEL
LIN {X 0,Y 397.497,Z 497.542,A -85,B 0,C 180,E1 -11228.185,E2 -11228.185} C_VEL
LIN {X 0,Y 400.964,Z 513.426,A -85,B 0,C 180,E1 -11228.768,E2 -11228.768} C_VEL
LIN {X 0,Y 403.05,Z 526.4,A -85,B 0,C 180,E1 -11229.389,E2 -11229.389} C_VEL
LIN {X 0,Y 403.627,Z 533.089,A -85,B 0,C 180,E1 -11229.754,E2 -11229.754} C_VEL
LIN {X 0,Y 402.795,Z 545.937,A -85,B 0,C 180,E1 -11230.508,E2 -11230.508} C_VEL
LIN {X 0,Y 401.736,Z 559.198,A -85,B 0,C 180,E1 -11231.515,E2 -11231.515} C_VEL
LIN {X 0,Y 400.549,Z 571.09,A -85,B 0,C 180,E1 -11232.647,E2 -11232.647} C_VEL
LIN {X 0,Y 399.463,Z 581.928,A -85,B 0,C 180,E1 -11233.914,E2 -11233.914} C_VEL
LIN {X 0,Y 398.451,Z 592.616,A -85,B 0,C 180,E1 -11235.444,E2 -11235.444} C_VEL
LIN {X 0,Y 397.633,Z 601.417,A -85,B 0,C 180,E1 -11236.978,E2 -11236.978} C_VEL
LIN {X 0,Y 397.017,Z 608.719,A -85,B 0,C 180,E1 -11238.514,E2 -11238.514} C_VEL
LIN {X 0,Y 396.443,Z 615.684,A -85,B 0,C 180,E1 -11240.306,E2 -11240.306} C_VEL
LIN {X 0,Y 396.03,Z 621.916,A -85,B 0,C 180,E1 -11242.353,E2 -11242.353} C_VEL
LIN {X 0,Y 395.908,Z 625.454,A -85,B 0,C 180,E1 -11243.887,E2 -11243.887} C_VEL
LIN {X 0,Y 395.779,Z 628.898,A -85,B 0,C 180,E1 -11245.928,E2 -11245.928} C_VEL
LIN {X 0,Y 395.782,Z 630.934,A -85,B 0,C 180,E1 -11247.966,E2 -11247.966} C_VEL
LIN {X 0,Y 395.778,Z 631.609,A -85,B 0,C 180,E1 -11250.001,E2 -11250.001} C_VEL
LIN {X 0,Y 395.788,Z 630.927,A -85,B 0,C 180,E1 -11252.036,E2 -11252.036} C_VEL
LIN {X 0,Y 395.78,Z 628.884,A -85,B 0,C 180,E1 -11254.074,E2 -11254.074} C_VEL
LIN {X 0,Y 395.91,Z 625.436,A -85,B 0,C 180,E1 -11256.115,E2 -11256.115} C_VEL
LIN {X 0,Y 396.088,Z 620.476,A -85,B 0,C 180,E1 -11258.162,E2 -11258.162} C_VEL
LIN {X 0,Y 396.448,Z 615.658,A -85,B 0,C 180,E1 -11259.697,E2 -11259.697} C_VEL
LIN {X 0,Y 397.007,Z 608.684,A -85,B 0,C 180,E1 -11261.489,E2 -11261.489} C_VEL
LIN {X 0,Y 397.609,Z 601.374,A -85,B 0,C 180,E1 -11263.026,E2 -11263.026} C_VEL
LIN {X 0,Y 398.467,Z 592.563,A -85,B 0,C 180,E1 -11264.558,E2 -11264.558} C_VEL
LIN {X 0,Y 399.525,Z 581.864,A -85,B 0,C 180,E1 -11266.086,E2 -11266.086} C_VEL
LIN {X 0,Y 400.583,Z 571.011,A -85,B 0,C 180,E1 -11267.354,E2 -11267.354} C_VEL
LIN {X 0,Y 401.706,Z 559.097,A -85,B 0,C 180,E1 -11268.489,E2 -11268.489} C_VEL
LIN {X 0,Y 402.758,Z 546.627,A -85,B 0,C 180,E1 -11269.44,E2 -11269.44} C_VEL
LIN {X 0,Y 403.884,Z 532.175,A -85,B 0,C 180,E1 -11270.367,E2 -11270.367} C_VEL
LIN {X 0,Y 402.58,Z 518.403,A -85,B 0,C 180,E1 -11271.246,E2 -11271.246} C_VEL
LIN {X 0,Y 400.059,Z 505.877,A -85,B 0,C 180,E1 -11271.983,E2 -11271.983} C_VEL
LIN {X 0,Y 397.854,Z 497.556,A -85,B 0,C 180,E1 -11272.458,E2 -11272.458} C_VEL
LIN {X 0,Y 398.792,Z 488.507,A -85,B 0,C 180,E1 -11276.142,E2 -11276.142} C_VEL
LIN {X 0,Y 399.966,Z 481.05,A -85,B 0,C 180,E1 -11279.473,E2 -11279.473} C_VEL
LIN {X 0,Y 401.17,Z 475.45,A -85,B 0,C 180,E1 -11282.258,E2 -11282.258} C_VEL
LIN {X 0,Y 401.515,Z 472.317,A -85,B 0,C 180,E1 -11284.065,E2 -11284.065} C_VEL
LIN {X 0,Y 401.039,Z 468.819,A -85,B 0,C 180,E1 -11286.573,E2 -11286.573} C_VEL
LIN {X 0,Y 400.481,Z 465.736,A -85,B 0,C 180,E1 -11289.452,E2 -11289.452} C_VEL
LIN {X 0,Y 400.117,Z 463.924,A -85,B 0,C 180,E1 -11291.873,E2 -11291.873} C_VEL
LIN {X 0,Y 399.815,Z 462.72,A -85,B 0,C 180,E1 -11294.68,E2 -11294.68} C_VEL
LIN {X 0,Y 399.723,Z 462.446,A -85,B 0,C 180,E1 -11297.601,E2 -11297.601} C_VEL
LIN {X 0,Y 399.734,Z 463.214,A -85,B 0,C 180,E1 -11300.733,E2 -11300.733} C_VEL
LIN {X 0,Y 399.703,Z 464.57,A -85,B 0,C 180,E1 -11303.286,E2 -11303.286} C_VEL
LIN {X 0,Y 399.318,Z 466.544,A -85,B 0,C 180,E1 -11305.814,E2 -11305.814} C_VEL
LIN {X 0,Y 398.557,Z 469.974,A -85,B 0,C 180,E1 -11309.245,E2 -11309.245} C_VEL
LIN {X 0,Y 397.989,Z 473.987,A -85,B 0,C 180,E1 -11312.669,E2 -11312.669} C_VEL
LIN {X 0,Y 397.451,Z 478.359,A -85,B 0,C 180,E1 -11316.002,E2 -11316.002} C_VEL
LIN {X 0,Y 397.103,Z 482.957,A -85,B 0,C 180,E1 -11319.27,E2 -11319.27} C_VEL
LIN {X 0,Y 396.986,Z 484.42,A -85,B 0,C 180,E1 -11320.269,E2 -11320.269} C_VEL
LIN {X 0,Y 401.249,Z 497.93,A -85,B 0,C 180,E1 -11321.283,E2 -11321.283} C_VEL
LIN {X 0,Y 403.498,Z 507.842,A -85,B 0,C 180,E1 -11322.058,E2 -11322.058} C_VEL
LIN {X 0,Y 403.864,Z 511.546,A -85,B 0,C 180,E1 -11322.345,E2 -11322.345} C_VEL
LIN {X 0,Y 402.684,Z 523.896,A -85,B 0,C 180,E1 -11323.263,E2 -11323.263} C_VEL
LIN {X 0,Y 401.497,Z 536.201,A -85,B 0,C 180,E1 -11324.428,E2 -11324.428} C_VEL
LIN {X 0,Y 400.241,Z 547.698,A -85,B 0,C 180,E1 -11325.769,E2 -11325.769} C_VEL
LIN {X 0,Y 399.247,Z 556.478,A -85,B 0,C 180,E1 -11327.03,E2 -11327.03} C_VEL
LIN {X 0,Y 398.331,Z 565.145,A -85,B 0,C 180,E1 -11328.551,E2 -11328.551} C_VEL
LIN {X 0,Y 397.629,Z 572.245,A -85,B 0,C 180,E1 -11330.077,E2 -11330.077} C_VEL
LIN {X 0,Y 396.904,Z 578.85,A -85,B 0,C 180,E1 -11331.856,E2 -11331.856} C_VEL
LIN {X 0,Y 396.577,Z 582.978,A -85,B 0,C 180,E1 -11333.287,E2 -11333.287} C_VEL
LIN {X 0,Y 396.158,Z 586.538,A -85,B 0,C 180,E1 -11334.911,E2 -11334.911} C_VEL
LIN {X 0,Y 396.202,Z 588.157,A -85,B 0,C 180,E1 -11335.931,E2 -11335.931} C_VEL
LIN {X 0,Y 396.08,Z 589.388,A -85,B 0,C 180,E1 -11336.949,E2 -11336.949} C_VEL
LIN {X 0,Y 395.947,Z 590.227,A -85,B 0,C 180,E1 -11337.966,E2 -11337.966} C_VEL
LIN {X 0,Y 395.868,Z 590.646,A -85,B 0,C 180,E1 -11338.983,E2 -11338.983} C_VEL
LIN {X 0,Y 395.841,Z 590.632,A -85,B 0,C 180,E1 -11340,E2 -11340} C_VEL
LIN {X 0,Y 395.936,Z 589.409,A -85,B 0,C 180,E1 -11342.035,E2 -11342.035} C_VEL
LIN {X 0,Y 395.996,Z 588.175,A -85,B 0,C 180,E1 -11343.052,E2 -11343.052} C_VEL
LIN {X 0,Y 396.018,Z 585.523,A -85,B 0,C 180,E1 -11344.581,E2 -11344.581} C_VEL
LIN {X 0,Y 396.236,Z 581.844,A -85,B 0,C 180,E1 -11346.109,E2 -11346.109} C_VEL
LIN {X 0,Y 396.439,Z 577.052,A -85,B 0,C 180,E1 -11347.641,E2 -11347.641} C_VEL
LIN {X 0,Y 396.944,Z 569.855,A -85,B 0,C 180,E1 -11349.426,E2 -11349.426} C_VEL
LIN {X 0,Y 397.487,Z 562.129,A -85,B 0,C 180,E1 -11350.957,E2 -11350.957} C_VEL
LIN {X 0,Y 398.077,Z 554.31,A -85,B 0,C 180,E1 -11352.231,E2 -11352.231} C_VEL
LIN {X 0,Y 398.958,Z 543.835,A -85,B 0,C 180,E1 -11353.628,E2 -11353.628} C_VEL
LIN {X 0,Y 399.699,Z 532.728,A -85,B 0,C 180,E1 -11354.833,E2 -11354.833} C_VEL
LIN {X 0,Y 400.447,Z 521.903,A -85,B 0,C 180,E1 -11355.785,E2 -11355.785} C_VEL
LIN {X 0,Y 401.261,Z 508.485,A -85,B 0,C 180,E1 -11356.709,E2 -11356.709} C_VEL
LIN {X 0,Y 399.88,Z 499.721,A -85,B 0,C 180,E1 -11357.253,E2 -11357.253} C_VEL
LIN {X 0,Y 396.93,Z 485.188,A -85,B 0,C 180,E1 -11357.983,E2 -11357.983} C_VEL
LIN {X 0,Y 396.322,Z 481.908,A -85,B 0,C 180,E1 -11358.129,E2 -11358.129} C_VEL
LIN {X 0,Y 396.431,Z 477.386,A -85,B 0,C 180,E1 -11360.767,E2 -11360.767} C_VEL
LIN {X 0,Y 396.632,Z 471.843,A -85,B 0,C 180,E1 -11364.051,E2 -11364.051} C_VEL
LIN {X 0,Y 396.941,Z 465.767,A -85,B 0,C 180,E1 -11367.714,E2 -11367.714} C_VEL
LIN {X 0,Y 397.131,Z 460.64,A -85,B 0,C 180,E1 -11370.878,E2 -11370.878} C_VEL
LIN {X 0,Y 397.383,Z 454.959,A -85,B 0,C 180,E1 -11374.468,E2 -11374.468} C_VEL
LIN {X 0,Y 397.348,Z 450.673,A -85,B 0,C 180,E1 -11377.256,E2 -11377.256} C_VEL
LIN {X 0,Y 397.19,Z 449.637,A -85,B 0,C 180,E1 -11377.992,E2 -11377.992} C_VEL
LIN {X 0,Y 397.095,Z 449.646,A -85,B 0,C 180,E1 -11380.908,E2 -11380.908} C_VEL
LIN {X 0,Y 397.109,Z 449.647,A -85,B 0,C 180,E1 -11383.648,E2 -11383.648} C_VEL
LIN {X 0,Y 397.11,Z 449.651,A -85,B 0,C 180,E1 -11386.52,E2 -11386.52} C_VEL
LIN {X 0,Y 397.162,Z 449.759,A -85,B 0,C 180,E1 -11388.594,E2 -11388.594} C_VEL
LIN {X 0,Y 397.983,Z 454.771,A -85,B 0,C 180,E1 -11390.987,E2 -11390.987} C_VEL
LIN {X 0,Y 398.07,Z 459.35,A -85,B 0,C 180,E1 -11393.109,E2 -11393.109} C_VEL
LIN {X 0,Y 397.818,Z 465.943,A -85,B 0,C 180,E1 -11396.132,E2 -11396.132} C_VEL
LIN {X 0,Y 397.551,Z 472.589,A -85,B 0,C 180,E1 -11399.157,E2 -11399.157} C_VEL
LIN {X 0,Y 397.296,Z 480.35,A -85,B 0,C 180,E1 -11402.616,E2 -11402.616} C_VEL
LIN {X 0,Y 397.038,Z 488.156,A -85,B 0,C 180,E1 -11405.974,E2 -11405.974} C_VEL
LIN {X 0,Y 396.951,Z 493.091,A -85,B 0,C 180,E1 -11407.986,E2 -11407.986} C_VEL
LIN {X 0,Y 400.887,Z 508.323,A -85,B 0,C 180,E1 -11408.616,E2 -11408.616} C_VEL
LIN {X 0,Y 403.624,Z 521.993,A -85,B 0,C 180,E1 -11409.338,E2 -11409.338} C_VEL
LIN {X 0,Y 404.208,Z 527.261,A -85,B 0,C 180,E1 -11409.65,E2 -11409.65} C_VEL
LIN {X 0,Y 403.308,Z 540.672,A -85,B 0,C 180,E1 -11410.461,E2 -11410.461} C_VEL
LIN {X 0,Y 402.337,Z 552.879,A -85,B 0,C 180,E1 -11411.409,E2 -11411.409} C_VEL
LIN {X 0,Y 401.069,Z 564.657,A -85,B 0,C 180,E1 -11412.536,E2 -11412.536} C_VEL
LIN {X 0,Y 400.187,Z 574.46,A -85,B 0,C 180,E1 -11413.68,E2 -11413.68} C_VEL
LIN {X 0,Y 399.015,Z 585.252,A -85,B 0,C 180,E1 -11415.202,E2 -11415.202} C_VEL
LIN {X 0,Y 398.165,Z 594.168,A -85,B 0,C 180,E1 -11416.733,E2 -11416.733} C_VEL
LIN {X 0,Y 397.233,Z 602.693,A -85,B 0,C 180,E1 -11418.518,E2 -11418.518} C_VEL
LIN {X 0,Y 396.628,Z 609.569,A -85,B 0,C 180,E1 -11420.308,E2 -11420.308} C_VEL
LIN {X 0,Y 396.162,Z 615.732,A -85,B 0,C 180,E1 -11422.353,E2 -11422.353} C_VEL
LIN {X 0,Y 395.999,Z 619.235,A -85,B 0,C 180,E1 -11423.886,E2 -11423.886} C_VEL
LIN {X 0,Y 395.78,Z 622.656,A -85,B 0,C 180,E1 -11425.926,E2 -11425.926} C_VEL
LIN {X 0,Y 395.757,Z 624.693,A -85,B 0,C 180,E1 -11427.963,E2 -11427.963} C_VEL
LIN {X 0,Y 395.759,Z 625.396,A -85,B 0,C 180,E1 -11429.999,E2 -11429.999} C_VEL
LIN {X 0,Y 395.755,Z 624.769,A -85,B 0,C 180,E1 -11432.034,E2 -11432.034} C_VEL
LIN {X 0,Y 395.779,Z 622.797,A -85,B 0,C 180,E1 -11434.072,E2 -11434.072} C_VEL
LIN {X 0,Y 395.977,Z 619.438,A -85,B 0,C 180,E1 -11436.112,E2 -11436.112} C_VEL
LIN {X 0,Y 396.204,Z 614.974,A -85,B 0,C 180,E1 -11438.017,E2 -11438.017} C_VEL
LIN {X 0,Y 395.687,Z 612.788,A -85,B 0,C 180,E1 -11438.806,E2 -11438.806} C_VEL
LIN {X 0,Y 393.13,Z 608.893,A -85,B 0,C 180,E1 -11440.08,E2 -11440.08} C_VEL
LIN {X 0,Y 390.724,Z 604.553,A -85,B 0,C 180,E1 -11441.334,E2 -11441.334} C_VEL
LIN {X 0,Y 390.448,Z 601.498,A -85,B 0,C 180,E1 -11442.08,E2 -11442.08} C_VEL
LIN {X 0,Y 391.201,Z 593.608,A -85,B 0,C 180,E1 -11443.726,E2 -11443.726} C_VEL
LIN {X 0,Y 392.213,Z 584.304,A -85,B 0,C 180,E1 -11445.324,E2 -11445.324} C_VEL
LIN {X 0,Y 393.349,Z 574.256,A -85,B 0,C 180,E1 -11446.743,E2 -11446.743} C_VEL
LIN {X 0,Y 394.551,Z 563.2,A -85,B 0,C 180,E1 -11448.027,E2 -11448.027} C_VEL
LIN {X 0,Y 395.742,Z 551.021,A -85,B 0,C 180,E1 -11449.179,E2 -11449.179} C_VEL
LIN {X 0,Y 396.837,Z 537.763,A -85,B 0,C 180,E1 -11450.176,E2 -11450.176} C_VEL
LIN {X 0,Y 397.376,Z 526.14,A -85,B 0,C 180,E1 -11450.876,E2 -11450.876} C_VEL
LIN {X 0,Y 394.974,Z 513.06,A -85,B 0,C 180,E1 -11451.637,E2 -11451.637} C_VEL
LIN {X 0,Y 391.448,Z 498.57,A -85,B 0,C 180,E1 -11452.314,E2 -11452.314} C_VEL
LIN {X 0,Y 389.908,Z 492.936,A -85,B 0,C 180,E1 -11452.567,E2 -11452.567} C_VEL
LIN {X 0,Y 390.192,Z 484.389,A -85,B 0,C 180,E1 -11456.192,E2 -11456.192} C_VEL
LIN {X 0,Y 390.479,Z 476.578,A -85,B 0,C 180,E1 -11459.662,E2 -11459.662} C_VEL
LIN {X 0,Y 390.736,Z 468.708,A -85,B 0,C 180,E1 -11463.268,E2 -11463.268} C_VEL
LIN {X 0,Y 391.023,Z 462.049,A -85,B 0,C 180,E1 -11466.377,E2 -11466.377} C_VEL
LIN {X 0,Y 391.106,Z 456.442,A -85,B 0,C 180,E1 -11468.969,E2 -11468.969} C_VEL
LIN {X 0,Y 390.139,Z 450.517,A -85,B 0,C 180,E1 -11471.87,E2 -11471.87} C_VEL
LIN {X 0,Y 390.112,Z 450.518,A -85,B 0,C 180,E1 -11475.364,E2 -11475.364} C_VEL
LIN {X 0,Y 390.098,Z 450.52,A -85,B 0,C 180,E1 -11478.195,E2 -11478.195} C_VEL
LIN {X 0,Y 390.087,Z 450.519,A -85,B 0,C 180,E1 -11480.907,E2 -11480.907} C_VEL
LIN {X 0,Y 390.077,Z 450.519,A -85,B 0,C 180,E1 -11484.792,E2 -11484.792} C_VEL
LIN {X 0,Y 390.04,Z 450.52,A -85,B 0,C 180,E1 -11488.497,E2 -11488.497} C_VEL
LIN {X 0,Y 390.108,Z 450.514,A -85,B 0,C 180,E1 -11492.069,E2 -11492.069} C_VEL
LIN {X 0,Y 390.072,Z 450.522,A -85,B 0,C 180,E1 -11495.519,E2 -11495.519} C_VEL
LIN {X 0,Y 390.083,Z 450.513,A -85,B 0,C 180,E1 -11498.879,E2 -11498.879} C_VEL
LIN {X 0,Y 390.121,Z 450.514,A -85,B 0,C 180,E1 -11502.166,E2 -11502.166} C_VEL
LIN {X 0,Y 390.139,Z 450.511,A -85,B 0,C 180,E1 -11505.392,E2 -11505.392} C_VEL
LIN {X 0,Y 390.15,Z 450.507,A -85,B 0,C 180,E1 -11508.571,E2 -11508.571} C_VEL
LIN {X 0,Y 390.333,Z 450.484,A -85,B 0,C 180,E1 -11511.992,E2 -11511.992} C_VEL
LIN {X 0,Y 390.226,Z 450.498,A -85,B 0,C 180,E1 -11514.833,E2 -11514.833} C_VEL
LIN {X 0,Y 390.41,Z 450.476,A -85,B 0,C 180,E1 -11517.937,E2 -11517.937} C_VEL
LIN {X 0,Y 390.541,Z 450.462,A -85,B 0,C 180,E1 -11520,E2 -11520} C_VEL
LIN {X 0,Y 390.306,Z 450.474,A -85,B 0,C 180,E1 -11523.096,E2 -11523.096} C_VEL
LIN {X 0,Y 390.319,Z 450.488,A -85,B 0,C 180,E1 -11526.202,E2 -11526.202} C_VEL
LIN {X 0,Y 390.304,Z 450.49,A -85,B 0,C 180,E1 -11528.282,E2 -11528.282} C_VEL
LIN {X 0,Y 390.168,Z 450.503,A -85,B 0,C 180,E1 -11532.483,E2 -11532.483} C_VEL
LIN {X 0,Y 390.129,Z 450.508,A -85,B 0,C 180,E1 -11535.677,E2 -11535.677} C_VEL
LIN {X 0,Y 390.095,Z 450.514,A -85,B 0,C 180,E1 -11538.923,E2 -11538.923} C_VEL
LIN {X 0,Y 390.03,Z 450.525,A -85,B 0,C 180,E1 -11542.235,E2 -11542.235} C_VEL
LIN {X 0,Y 390.109,Z 450.517,A -85,B 0,C 180,E1 -11545.744,E2 -11545.744} C_VEL
LIN {X 0,Y 390.056,Z 450.526,A -85,B 0,C 180,E1 -11549.11,E2 -11549.11} C_VEL
LIN {X 0,Y 390.034,Z 450.526,A -85,B 0,C 180,E1 -11552.722,E2 -11552.722} C_VEL
LIN {X 0,Y 390.049,Z 450.525,A -85,B 0,C 180,E1 -11555.827,E2 -11555.827} C_VEL
LIN {X 0,Y 390.066,Z 450.522,A -85,B 0,C 180,E1 -11559.22,E2 -11559.22} C_VEL
LIN {X 0,Y 390.113,Z 450.516,A -85,B 0,C 180,E1 -11562.388,E2 -11562.388} C_VEL
LIN {X 0,Y 390.054,Z 450.523,A -85,B 0,C 180,E1 -11565.358,E2 -11565.358} C_VEL
LIN {X 0,Y 390.103,Z 450.645,A -85,B 0,C 180,E1 -11568.994,E2 -11568.994} C_VEL
LIN {X 0,Y 391.507,Z 458.061,A -85,B 0,C 180,E1 -11572.388,E2 -11572.388} C_VEL
LIN {X 0,Y 393.009,Z 466.037,A -85,B 0,C 180,E1 -11575.876,E2 -11575.876} C_VEL
LIN {X 0,Y 393.035,Z 470.162,A -85,B 0,C 180,E1 -11577.56,E2 -11577.56} C_VEL
LIN {X 0,Y 392.186,Z 477.62,A -85,B 0,C 180,E1 -11580.477,E2 -11580.477} C_VEL
LIN {X 0,Y 391.322,Z 486.55,A -85,B 0,C 180,E1 -11583.894,E2 -11583.894} C_VEL
LIN {X 0,Y 390.582,Z 495.504,A -85,B 0,C 180,E1 -11587.242,E2 -11587.242} C_VEL
LIN {X 0,Y 390.481,Z 496.853,A -85,B 0,C 180,E1 -11587.742,E2 -11587.742} C_VEL
LIN {X 0,Y 394.327,Z 514.502,A -85,B 0,C 180,E1 -11588.425,E2 -11588.425} C_VEL
LIN {X 0,Y 396.335,Z 527.437,A -85,B 0,C 180,E1 -11589.071,E2 -11589.071} C_VEL
LIN {X 0,Y 396.936,Z 533.337,A -85,B 0,C 180,E1 -11589.412,E2 -11589.412} C_VEL
LIN {X 0,Y 396.068,Z 546.288,A -85,B 0,C 180,E1 -11590.189,E2 -11590.189} C_VEL
LIN {X 0,Y 395.002,Z 559.161,A -85,B 0,C 180,E1 -11591.188,E2 -11591.188} C_VEL
LIN {X 0,Y 393.764,Z 571.048,A -85,B 0,C 180,E1 -11592.338,E2 -11592.338} C_VEL
LIN {X 0,Y 392.615,Z 581.883,A -85,B 0,C 180,E1 -11593.626,E2 -11593.626} C_VEL
LIN {X 0,Y 391.523,Z 592.568,A -85,B 0,C 180,E1 -11595.181,E2 -11595.181} C_VEL
LIN {X 0,Y 390.646,Z 601.367,A -85,B 0,C 180,E1 -11596.741,E2 -11596.741} C_VEL
LIN {X 0,Y 390.04,Z 608.668,A -85,B 0,C 180,E1 -11598.306,E2 -11598.306} C_VEL
LIN {X 0,Y 389.394,Z 615.631,A -85,B 0,C 180,E1 -11600.129,E2 -11600.129} C_VEL
LIN {X 0,Y 388.959,Z 621.862,A -85,B 0,C 180,E1 -11602.213,E2 -11602.213} C_VEL
LIN {X 0,Y 388.832,Z 625.4,A -85,B 0,C 180,E1 -11603.776,E2 -11603.776} C_VEL
LIN {X 0,Y 388.703,Z 628.844,A -85,B 0,C 180,E1 -11605.854,E2 -11605.854} C_VEL
LIN {X 0,Y 388.678,Z 630.878,A -85,B 0,C 180,E1 -11607.929,E2 -11607.929} C_VEL
LIN {X 0,Y 388.689,Z 631.553,A -85,B 0,C 180,E1 -11610.001,E2 -11610.001} C_VEL
LIN {X 0,Y 388.683,Z 630.871,A -85,B 0,C 180,E1 -11612.074,E2 -11612.074} C_VEL
LIN {X 0,Y 388.704,Z 628.828,A -85,B 0,C 180,E1 -11614.149,E2 -11614.149} C_VEL
LIN {X 0,Y 388.834,Z 625.38,A -85,B 0,C 180,E1 -11616.227,E2 -11616.227} C_VEL
LIN {X 0,Y 389.037,Z 620.42,A -85,B 0,C 180,E1 -11618.311,E2 -11618.311} C_VEL
LIN {X 0,Y 389.396,Z 615.602,A -85,B 0,C 180,E1 -11619.874,E2 -11619.874} C_VEL
LIN {X 0,Y 390.033,Z 608.629,A -85,B 0,C 180,E1 -11621.697,E2 -11621.697} C_VEL
LIN {X 0,Y 390.644,Z 601.32,A -85,B 0,C 180,E1 -11623.262,E2 -11623.262} C_VEL
LIN {X 0,Y 391.543,Z 592.51,A -85,B 0,C 180,E1 -11624.821,E2 -11624.821} C_VEL
LIN {X 0,Y 392.658,Z 581.814,A -85,B 0,C 180,E1 -11626.375,E2 -11626.375} C_VEL
LIN {X 0,Y 393.793,Z 570.963,A -85,B 0,C 180,E1 -11627.663,E2 -11627.663} C_VEL
LIN {X 0,Y 394.97,Z 559.053,A -85,B 0,C 180,E1 -11628.816,E2 -11628.816} C_VEL
LIN {X 0,Y 396.624,Z 540.927,A -85,B 0,C 180,E1 -11630.215,E2 -11630.215} C_VEL
LIN {X 0,Y 397.279,Z 532.35,A -85,B 0,C 180,E1 -11630.791,E2 -11630.791} C_VEL
LIN {X 0,Y 396.133,Z 519.677,A -85,B 0,C 180,E1 -11631.641,E2 -11631.641} C_VEL
LIN {X 0,Y 393.791,Z 507.828,A -85,B 0,C 180,E1 -11632.391,E2 -11632.391} C_VEL
LIN {X 0,Y 390.959,Z 497.33,A -85,B 0,C 180,E1 -11633.047,E2 -11633.047} C_VEL
LIN {X 0,Y 391.981,Z 488.852,A -85,B 0,C 180,E1 -11636.632,E2 -11636.632} C_VEL
LIN {X 0,Y 393.243,Z 481.558,A -85,B 0,C 180,E1 -11640.028,E2 -11640.028} C_VEL
LIN {X 0,Y 394.273,Z 477.095,A -85,B 0,C 180,E1 -11642.329,E2 -11642.329} C_VEL
LIN {X 0,Y 394.662,Z 475.034,A -85,B 0,C 180,E1 -11643.508,E2 -11643.508} C_VEL
LIN {X 0,Y 394.531,Z 472.837,A -85,B 0,C 180,E1 -11644.973,E2 -11644.973} C_VEL
LIN {X 0,Y 394.053,Z 469.87,A -85,B 0,C 180,E1 -11647.331,E2 -11647.331} C_VEL
LIN {X 0,Y 393.59,Z 467.269,A -85,B 0,C 180,E1 -11650.004,E2 -11650.004} C_VEL
LIN {X 0,Y 393.178,Z 465.43,A -85,B 0,C 180,E1 -11652.873,E2 -11652.873} C_VEL
LIN {X 0,Y 392.941,Z 464.525,A -85,B 0,C 180,E1 -11655.77,E2 -11655.77} C_VEL
LIN {X 0,Y 392.873,Z 464.577,A -85,B 0,C 180,E1 -11658.707,E2 -11658.707} C_VEL
LIN {X 0,Y 392.901,Z 465.626,A -85,B 0,C 180,E1 -11661.912,E2 -11661.912} C_VEL
LIN {X 0,Y 392.786,Z 466.739,A -85,B 0,C 180,E1 -11663.81,E2 -11663.81} C_VEL
LIN {X 0,Y 392.281,Z 468.678,A -85,B 0,C 180,E1 -11666.263,E2 -11666.263} C_VEL
LIN {X 0,Y 391.545,Z 472.198,A -85,B 0,C 180,E1 -11669.829,E2 -11669.829} C_VEL
LIN {X 0,Y 390.894,Z 476.225,A -85,B 0,C 180,E1 -11673.29,E2 -11673.29} C_VEL
LIN {X 0,Y 390.396,Z 480.587,A -85,B 0,C 180,E1 -11676.669,E2 -11676.669} C_VEL
LIN {X 0,Y 390.08,Z 484.751,A -85,B 0,C 180,E1 -11679.669,E2 -11679.669} C_VEL
LIN {X 0,Y 394.513,Z 498.431,A -85,B 0,C 180,E1 -11680.765,E2 -11680.765} C_VEL
LIN {X 0,Y 396.948,Z 508.958,A -85,B 0,C 180,E1 -11681.649,E2 -11681.649} C_VEL
LIN {X 0,Y 397.367,Z 513.047,A -85,B 0,C 180,E1 -11681.982,E2 -11681.982} C_VEL
LIN {X 0,Y 396.072,Z 525.81,A -85,B 0,C 180,E1 -11682.976,E2 -11682.976} C_VEL
LIN {X 0,Y 394.803,Z 537.745,A -85,B 0,C 180,E1 -11684.157,E2 -11684.157} C_VEL
LIN {X 0,Y 393.457,Z 548.887,A -85,B 0,C 180,E1 -11685.518,E2 -11685.518} C_VEL
LIN {X 0,Y 392.403,Z 557.509,A -85,B 0,C 180,E1 -11686.8,E2 -11686.8} C_VEL
LIN {X 0,Y 391.436,Z 566.076,A -85,B 0,C 180,E1 -11688.347,E2 -11688.347} C_VEL
LIN {X 0,Y 390.689,Z 573.059,A -85,B 0,C 180,E1 -11689.899,E2 -11689.899} C_VEL
LIN {X 0,Y 389.927,Z 579.507,A -85,B 0,C 180,E1 -11691.71,E2 -11691.71} C_VEL
LIN {X 0,Y 389.54,Z 583.74,A -85,B 0,C 180,E1 -11693.238,E2 -11693.238} C_VEL
LIN {X 0,Y 389.1,Z 587.073,A -85,B 0,C 180,E1 -11694.819,E2 -11694.819} C_VEL
LIN {X 0,Y 389.132,Z 588.664,A -85,B 0,C 180,E1 -11695.857,E2 -11695.857} C_VEL
LIN {X 0,Y 389.026,Z 589.864,A -85,B 0,C 180,E1 -11696.893,E2 -11696.893} C_VEL
LIN {X 0,Y 388.883,Z 590.668,A -85,B 0,C 180,E1 -11697.929,E2 -11697.929} C_VEL
LIN {X 0,Y 388.797,Z 591.029,A -85,B 0,C 180,E1 -11698.964,E2 -11698.964} C_VEL
LIN {X 0,Y 388.768,Z 590.983,A -85,B 0,C 180,E1 -11700,E2 -11700} C_VEL
LIN {X 0,Y 388.871,Z 589.7,A -85,B 0,C 180,E1 -11702.072,E2 -11702.072} C_VEL
LIN {X 0,Y 388.901,Z 588.417,A -85,B 0,C 180,E1 -11703.108,E2 -11703.108} C_VEL
LIN {X 0,Y 388.951,Z 585.707,A -85,B 0,C 180,E1 -11704.664,E2 -11704.664} C_VEL
LIN {X 0,Y 389.157,Z 581.965,A -85,B 0,C 180,E1 -11706.221,E2 -11706.221} C_VEL
LIN {X 0,Y 389.383,Z 577.098,A -85,B 0,C 180,E1 -11707.78,E2 -11707.78} C_VEL
